PROGRAM MAIN
VAR
	//==============================================================
	// EN: Main machine control function blocks
	// PT: Blocos principais de controle da máquina
	//==============================================================
	instFBSlitter1Control              : FB_SlitterControl;
	instFB_RotaryKnife                 : FB_RotaryKnife;
	// instFB_MetricsAndCalculation    : FB_MetricsAndCalculation;
	instFB_PaperDirectionControl       : FB_PaperDirectionControl;
	instFB_AutomaticOrderChange_V1     : FB_AutomaticOrderChange_V1;
	instFB_AlarmControl                : FB_AlarmControl;
	instFBSavePersistentData           : FB_SavePersistentData;

	//==============================================================
	// EN: Stacker control function blocks
	// PT: Blocos de controle dos empilhadores
	//==============================================================
	instFBLowerStackerControl          : FB_SimpleSheetStackerControl;
	instFBLowerStackerControlV1        : FB_SimpleSheetStackerControl_1;
	instFBUpperStackerControl          : FB_ComplexSheetStackerControl;

	//==============================================================
	// EN: Persistent data control status
	// PT: Estado do controle de dados persistentes
	//==============================================================
	bStart                             : BOOL;
	bError                             : BOOL;
	bBusy                              : BOOL;
	nErrorId                           : UDINT;
	fbR_Trig                           : R_TRIG;

	//==============================================================
	// EN: Machine interlock and control signals
	// PT: Sinais de intertravamento e controle da máquina
	//==============================================================
	slitterHomeComplete                : BOOL;
	aocReferenceSwitch                 : BOOL;
	lineSpeedUpFromAOC                 : BOOL;
	lineSpeedDownFromAOC               : BOOL;
	lineStopFromAOC                    : BOOL;
	executePositioningFromAOC          : BOOL;
	rotaryKnifeSpeedRefFromAOC         : LREAL;
	slitterSpeedRefFromAOC             : LREAL;
	lineStopFromRotaryKnife            : BOOL;
	lineStopFromSlitter                : BOOL;
	lineStopFromLowerStacker           : BOOL;
	aocRunning                         : BOOL;

	//==============================================================
	// EN: Program initialization
	// PT: Inicialização do programa
	//==============================================================
	firstScan                          : BOOL := TRUE;
	lineStopFromUpperStacker: BOOL;
END_VAR

//==============================================================
// EN: Cyclic machine control sequence
// PT: Sequência cíclica de controle da máquina
//==============================================================
_00_UpdateHardware();
_01_SlitterControl();
_02_RotaryKnifeControl();
_04_AutomaticOrderChange();
_05_LineControl();
_06_AlarmsControl();
_07_LowerStackerControl();
_08_UpperStackerControl();

// EN: Publish the upper stacker alarms and include them in the general indication.
// PT: Publica os alarmes do stacker superior e os inclui na indicação geral.
hmiAlarms.upperStacker :=
	instFBUpperStackerControl.hmiAlarms;

hmiStatus.alarmActive :=
	hmiStatus.alarmActive OR
	instFBUpperStackerControl.alarmActive;

// EN: Update persistent data management.
// PT: Atualiza o gerenciamento dos dados persistentes.
instFBSavePersistentData();

// EN: Apply default commands during the first PLC scan.
// PT: Aplica os comandos padrão durante o primeiro ciclo do PLC.
IF firstScan THEN
	hmiCommands.lowerStacker.backstopAutoCmd := TRUE;
	hmiCommands.lowerStacker.conveyorLevelerAutoCmd := TRUE;

	hmiCommands.upperStacker.backstopAutoCmd := TRUE;
	hmiCommands.upperStacker.elevatorAutoCmd := TRUE;

END_IF

firstScan := FALSE;

(*==============================================================================================================================
CPNTeck - Automação industrial
(c)Copyright 2023 All Rights Reserved
_______________________________________________________________________________________________________________________________
Library: <N/A or library name>
Tested with: <PLC / IPC model>
Engineering: <TwinCAT version>
Restrictions: <text>
Requirements: <text>
Functionality: <short description>
Support: <email>
Note: Parameter comments are only available in language 'English (United States)'
_______________________________________________________________________________________________________________________________
Change log table:

Version  		| Date        			| Expert in charge  	| Changes applied
<xx.xx.xx>		| <dd.mm.yyyy>  		| <name>              | <changes>

===============================================================================================================================*)

METHOD _00_UpdateHardware
VAR_INPUT
END_VAR

SLT1_P1_100_UG1();
SLT1_P1_100_UG2();
SLT1_P1_100_UG3();
SLT1_P1_100_UG4();
SLT1_P1_100_UG5();

SLT1_P1_200_UG1();
SLT1_P1_200_UG2();
SLT1_P1_200_UG3();
SLT1_P1_200_UG4();
SLT1_P1_200_UG5();
SLT1_P1_200_UG6();
SLT1_P1_200_UG7();
SLT1_P1_200_UG8();


STK_P2_050_DI1();
STK_P2_050_DI2();
STK_P2_050_DO1();
STK_P2_050_DO2();
	
STK_P2_050_AO1();	
STK_P2_050_AO2();
STK_P2_050_AO3();
STK_P2_050_AO4();

STK_P2_050_ENC1();
//Io-Link master
STK_050_BC2();
//Io-Link Slaves

STKU_050_DIO1();	//Ch 0 - IO-Link IP67 Input/Output module
STKU_050_DIO2(); //Ch 1 - IO-Link DIN Rail Input/Output module
STKU_050_DIO3(); //Ch 1 - IO-Link DIN Rail Input/Output module


STKL_050_DIO1();	//Ch 0 - IO-Link IP67 Input/Output module
STKL_050_DIO2(); //Ch 1 - IO-Link DIN Rail Input/Output module
STKL_100_B01(); //Ch 2 - IO-Link Pile height sensor	

//CANOpen slave	
STKU_P2_100_UG8(enable := TRUE); //Backstop servo drive

// EN: Lift servo drive. Quick stop is generated by the elevator control block.
// PT: Servo do elevador. O quick stop é gerado pelo bloco de controle do elevador.
STKU_P2_100_UG9(enable := TRUE);

// Safety processor (TwinSAFE)
STK_P2_050_SP01(run := TRUE,
				 errorAcknowledgement := hmiCommands.slitter1.resetCmd OR hmiCommands.lowerStacker.resetCmd OR hmiCommands.upperStacker.resetCmd,
				 safetyReset := hmiCommands.slitter1.resetCmd OR hmiCommands.lowerStacker.resetCmd OR hmiCommands.upperStacker.resetCmd
);
END_METHOD

METHOD _01_SlitterControl
VAR_INPUT
END_VAR

//ARK_P1_050_AO02.Channel1
//ARK_P1_050_AO02.Channel3
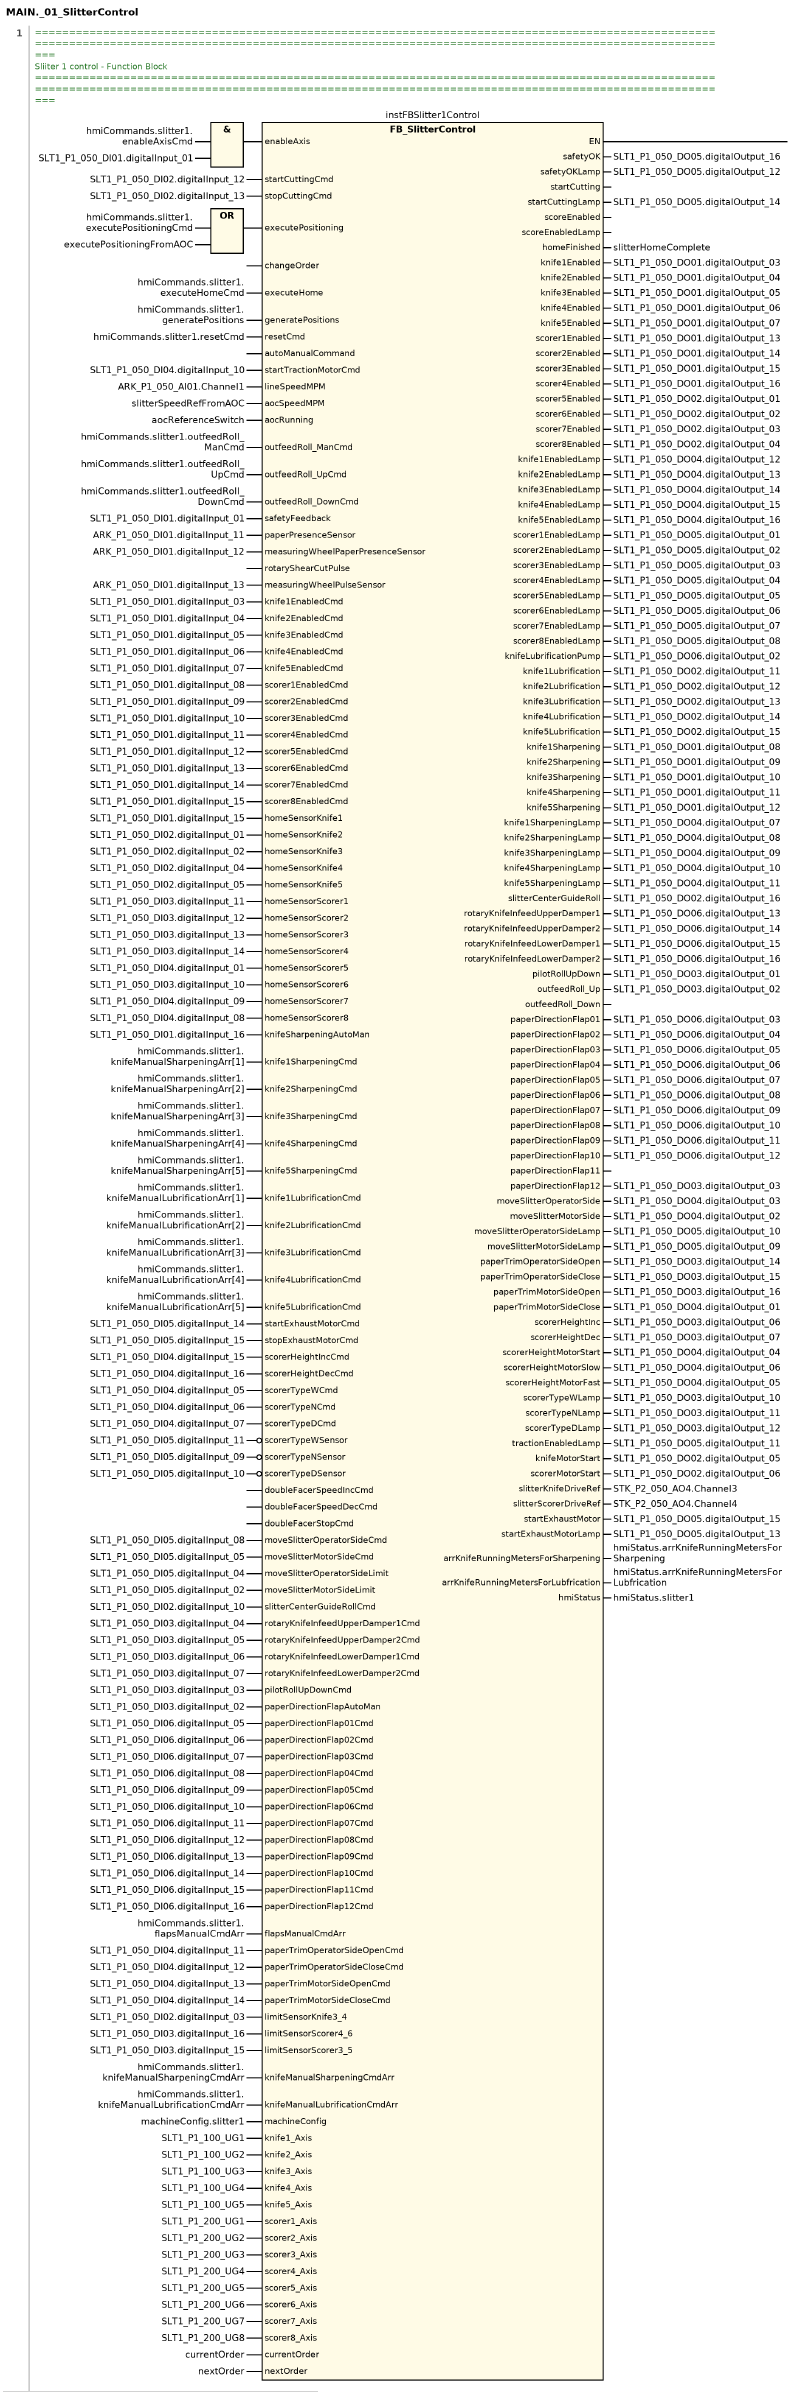
// NETWORK 1
// 					===========================================================================================================================================================================================================
//
// Sliiter 1 control - Function Block
//
// ===========================================================================================================================================================================================================
//
instFBSlitter1Control(
    enableAxis := hmiCommands.slitter1.enableAxisCmd AND SLT1_P1_050_DI01.digitalInput_01,
    startCuttingCmd := SLT1_P1_050_DI02.digitalInput_12,
    stopCuttingCmd := SLT1_P1_050_DI02.digitalInput_13,
    executePositioning := hmiCommands.slitter1.executePositioningCmd OR executePositioningFromAOC,
    executeHome := hmiCommands.slitter1.executeHomeCmd,
    generatePositions := hmiCommands.slitter1.generatePositions,
    resetCmd := hmiCommands.slitter1.resetCmd,
    startTractionMotorCmd := SLT1_P1_050_DI04.digitalInput_10,
    lineSpeedMPM := ARK_P1_050_AI01.Channel1,
    aocSpeedMPM := slitterSpeedRefFromAOC,
    aocRunning := aocReferenceSwitch,
    outfeedRoll_ManCmd := hmiCommands.slitter1.outfeedRoll_ManCmd,
    outfeedRoll_UpCmd := hmiCommands.slitter1.outfeedRoll_UpCmd,
    outfeedRoll_DownCmd := hmiCommands.slitter1.outfeedRoll_DownCmd,
    safetyFeedback := SLT1_P1_050_DI01.digitalInput_01,
    paperPresenceSensor := ARK_P1_050_DI01.digitalInput_11,
    measuringWheelPaperPresenceSensor := ARK_P1_050_DI01.digitalInput_12,
    measuringWheelPulseSensor := ARK_P1_050_DI01.digitalInput_13,
    knife1EnabledCmd := SLT1_P1_050_DI01.digitalInput_03,
    knife2EnabledCmd := SLT1_P1_050_DI01.digitalInput_04,
    knife3EnabledCmd := SLT1_P1_050_DI01.digitalInput_05,
    knife4EnabledCmd := SLT1_P1_050_DI01.digitalInput_06,
    knife5EnabledCmd := SLT1_P1_050_DI01.digitalInput_07,
    scorer1EnabledCmd := SLT1_P1_050_DI01.digitalInput_08,
    scorer2EnabledCmd := SLT1_P1_050_DI01.digitalInput_09,
    scorer3EnabledCmd := SLT1_P1_050_DI01.digitalInput_10,
    scorer4EnabledCmd := SLT1_P1_050_DI01.digitalInput_11,
    scorer5EnabledCmd := SLT1_P1_050_DI01.digitalInput_12,
    scorer6EnabledCmd := SLT1_P1_050_DI01.digitalInput_13,
    scorer7EnabledCmd := SLT1_P1_050_DI01.digitalInput_14,
    scorer8EnabledCmd := SLT1_P1_050_DI01.digitalInput_15,
    homeSensorKnife1 := SLT1_P1_050_DI01.digitalInput_15,
    homeSensorKnife2 := SLT1_P1_050_DI02.digitalInput_01,
    homeSensorKnife3 := SLT1_P1_050_DI02.digitalInput_02,
    homeSensorKnife4 := SLT1_P1_050_DI02.digitalInput_04,
    homeSensorKnife5 := SLT1_P1_050_DI02.digitalInput_05,
    homeSensorScorer1 := SLT1_P1_050_DI03.digitalInput_11,
    homeSensorScorer2 := SLT1_P1_050_DI03.digitalInput_12,
    homeSensorScorer3 := SLT1_P1_050_DI03.digitalInput_13,
    homeSensorScorer4 := SLT1_P1_050_DI03.digitalInput_14,
    homeSensorScorer5 := SLT1_P1_050_DI04.digitalInput_01,
    homeSensorScorer6 := SLT1_P1_050_DI03.digitalInput_10,
    homeSensorScorer7 := SLT1_P1_050_DI04.digitalInput_09,
    homeSensorScorer8 := SLT1_P1_050_DI04.digitalInput_08,
    knifeSharpeningAutoMan := SLT1_P1_050_DI01.digitalInput_16,
    knife1SharpeningCmd := hmiCommands.slitter1.knifeManualSharpeningArr[1],
    knife2SharpeningCmd := hmiCommands.slitter1.knifeManualSharpeningArr[2],
    knife3SharpeningCmd := hmiCommands.slitter1.knifeManualSharpeningArr[3],
    knife4SharpeningCmd := hmiCommands.slitter1.knifeManualSharpeningArr[4],
    knife5SharpeningCmd := hmiCommands.slitter1.knifeManualSharpeningArr[5],
    knife1LubrificationCmd := hmiCommands.slitter1.knifeManualLubrificationArr[1],
    knife2LubrificationCmd := hmiCommands.slitter1.knifeManualLubrificationArr[2],
    knife3LubrificationCmd := hmiCommands.slitter1.knifeManualLubrificationArr[3],
    knife4LubrificationCmd := hmiCommands.slitter1.knifeManualLubrificationArr[4],
    knife5LubrificationCmd := hmiCommands.slitter1.knifeManualLubrificationArr[5],
    startExhaustMotorCmd := SLT1_P1_050_DI05.digitalInput_14,
    stopExhaustMotorCmd := SLT1_P1_050_DI05.digitalInput_15,
    scorerHeightIncCmd := SLT1_P1_050_DI04.digitalInput_15,
    scorerHeightDecCmd := SLT1_P1_050_DI04.digitalInput_16,
    scorerTypeWCmd := SLT1_P1_050_DI04.digitalInput_05,
    scorerTypeNCmd := SLT1_P1_050_DI04.digitalInput_06,
    scorerTypeDCmd := SLT1_P1_050_DI04.digitalInput_07,
    scorerTypeWSensor := NOT SLT1_P1_050_DI05.digitalInput_11,
    scorerTypeNSensor := NOT SLT1_P1_050_DI05.digitalInput_09,
    scorerTypeDSensor := NOT SLT1_P1_050_DI05.digitalInput_10,
    moveSlitterOperatorSideCmd := SLT1_P1_050_DI05.digitalInput_08,
    moveSlitterMotorSideCmd := SLT1_P1_050_DI05.digitalInput_05,
    moveSlitterOperatorSideLimit := SLT1_P1_050_DI05.digitalInput_04,
    moveSlitterMotorSideLimit := SLT1_P1_050_DI05.digitalInput_02,
    slitterCenterGuideRollCmd := SLT1_P1_050_DI02.digitalInput_10,
    rotaryKnifeInfeedUpperDamper1Cmd := SLT1_P1_050_DI03.digitalInput_04,
    rotaryKnifeInfeedUpperDamper2Cmd := SLT1_P1_050_DI03.digitalInput_05,
    rotaryKnifeInfeedLowerDamper1Cmd := SLT1_P1_050_DI03.digitalInput_06,
    rotaryKnifeInfeedLowerDamper2Cmd := SLT1_P1_050_DI03.digitalInput_07,
    pilotRollUpDownCmd := SLT1_P1_050_DI03.digitalInput_03,
    paperDirectionFlapAutoMan := SLT1_P1_050_DI03.digitalInput_02,
    paperDirectionFlap01Cmd := SLT1_P1_050_DI06.digitalInput_05,
    paperDirectionFlap02Cmd := SLT1_P1_050_DI06.digitalInput_06,
    paperDirectionFlap03Cmd := SLT1_P1_050_DI06.digitalInput_07,
    paperDirectionFlap04Cmd := SLT1_P1_050_DI06.digitalInput_08,
    paperDirectionFlap05Cmd := SLT1_P1_050_DI06.digitalInput_09,
    paperDirectionFlap06Cmd := SLT1_P1_050_DI06.digitalInput_10,
    paperDirectionFlap07Cmd := SLT1_P1_050_DI06.digitalInput_11,
    paperDirectionFlap08Cmd := SLT1_P1_050_DI06.digitalInput_12,
    paperDirectionFlap09Cmd := SLT1_P1_050_DI06.digitalInput_13,
    paperDirectionFlap10Cmd := SLT1_P1_050_DI06.digitalInput_14,
    paperDirectionFlap11Cmd := SLT1_P1_050_DI06.digitalInput_15,
    paperDirectionFlap12Cmd := SLT1_P1_050_DI06.digitalInput_16,
    flapsManualCmdArr := hmiCommands.slitter1.flapsManualCmdArr,
    paperTrimOperatorSideOpenCmd := SLT1_P1_050_DI04.digitalInput_11,
    paperTrimOperatorSideCloseCmd := SLT1_P1_050_DI04.digitalInput_12,
    paperTrimMotorSideOpenCmd := SLT1_P1_050_DI04.digitalInput_13,
    paperTrimMotorSideCloseCmd := SLT1_P1_050_DI04.digitalInput_14,
    limitSensorKnife3_4 := SLT1_P1_050_DI02.digitalInput_03,
    limitSensorScorer4_6 := SLT1_P1_050_DI03.digitalInput_16,
    limitSensorScorer3_5 := SLT1_P1_050_DI03.digitalInput_15,
    knifeManualSharpeningCmdArr := hmiCommands.slitter1.knifeManualSharpeningCmdArr,
    knifeManualLubrificationCmdArr := hmiCommands.slitter1.knifeManualLubrificationCmdArr,
    machineConfig := machineConfig.slitter1,
    knife1_Axis := SLT1_P1_100_UG1,
    knife2_Axis := SLT1_P1_100_UG2,
    knife3_Axis := SLT1_P1_100_UG3,
    knife4_Axis := SLT1_P1_100_UG4,
    knife5_Axis := SLT1_P1_100_UG5,
    scorer1_Axis := SLT1_P1_200_UG1,
    scorer2_Axis := SLT1_P1_200_UG2,
    scorer3_Axis := SLT1_P1_200_UG3,
    scorer4_Axis := SLT1_P1_200_UG4,
    scorer5_Axis := SLT1_P1_200_UG5,
    scorer6_Axis := SLT1_P1_200_UG6,
    scorer7_Axis := SLT1_P1_200_UG7,
    scorer8_Axis := SLT1_P1_200_UG8,
    currentOrder := currentOrder,
    nextOrder := nextOrder,
    safetyOK => SLT1_P1_050_DO05.digitalOutput_16,
    safetyOKLamp => SLT1_P1_050_DO05.digitalOutput_12,
    startCuttingLamp => SLT1_P1_050_DO05.digitalOutput_14,
    homeFinished => slitterHomeComplete,
    knife1Enabled => SLT1_P1_050_DO01.digitalOutput_03,
    knife2Enabled => SLT1_P1_050_DO01.digitalOutput_04,
    knife3Enabled => SLT1_P1_050_DO01.digitalOutput_05,
    knife4Enabled => SLT1_P1_050_DO01.digitalOutput_06,
    knife5Enabled => SLT1_P1_050_DO01.digitalOutput_07,
    scorer1Enabled => SLT1_P1_050_DO01.digitalOutput_13,
    scorer2Enabled => SLT1_P1_050_DO01.digitalOutput_14,
    scorer3Enabled => SLT1_P1_050_DO01.digitalOutput_15,
    scorer4Enabled => SLT1_P1_050_DO01.digitalOutput_16,
    scorer5Enabled => SLT1_P1_050_DO02.digitalOutput_01,
    scorer6Enabled => SLT1_P1_050_DO02.digitalOutput_02,
    scorer7Enabled => SLT1_P1_050_DO02.digitalOutput_03,
    scorer8Enabled => SLT1_P1_050_DO02.digitalOutput_04,
    knife1EnabledLamp => SLT1_P1_050_DO04.digitalOutput_12,
    knife2EnabledLamp => SLT1_P1_050_DO04.digitalOutput_13,
    knife3EnabledLamp => SLT1_P1_050_DO04.digitalOutput_14,
    knife4EnabledLamp => SLT1_P1_050_DO04.digitalOutput_15,
    knife5EnabledLamp => SLT1_P1_050_DO04.digitalOutput_16,
    scorer1EnabledLamp => SLT1_P1_050_DO05.digitalOutput_01,
    scorer2EnabledLamp => SLT1_P1_050_DO05.digitalOutput_02,
    scorer3EnabledLamp => SLT1_P1_050_DO05.digitalOutput_03,
    scorer4EnabledLamp => SLT1_P1_050_DO05.digitalOutput_04,
    scorer5EnabledLamp => SLT1_P1_050_DO05.digitalOutput_05,
    scorer6EnabledLamp => SLT1_P1_050_DO05.digitalOutput_06,
    scorer7EnabledLamp => SLT1_P1_050_DO05.digitalOutput_07,
    scorer8EnabledLamp => SLT1_P1_050_DO05.digitalOutput_08,
    knifeLubrificationPump => SLT1_P1_050_DO06.digitalOutput_02,
    knife1Lubrification => SLT1_P1_050_DO02.digitalOutput_11,
    knife2Lubrification => SLT1_P1_050_DO02.digitalOutput_12,
    knife3Lubrification => SLT1_P1_050_DO02.digitalOutput_13,
    knife4Lubrification => SLT1_P1_050_DO02.digitalOutput_14,
    knife5Lubrification => SLT1_P1_050_DO02.digitalOutput_15,
    knife1Sharpening => SLT1_P1_050_DO01.digitalOutput_08,
    knife2Sharpening => SLT1_P1_050_DO01.digitalOutput_09,
    knife3Sharpening => SLT1_P1_050_DO01.digitalOutput_10,
    knife4Sharpening => SLT1_P1_050_DO01.digitalOutput_11,
    knife5Sharpening => SLT1_P1_050_DO01.digitalOutput_12,
    knife1SharpeningLamp => SLT1_P1_050_DO04.digitalOutput_07,
    knife2SharpeningLamp => SLT1_P1_050_DO04.digitalOutput_08,
    knife3SharpeningLamp => SLT1_P1_050_DO04.digitalOutput_09,
    knife4SharpeningLamp => SLT1_P1_050_DO04.digitalOutput_10,
    knife5SharpeningLamp => SLT1_P1_050_DO04.digitalOutput_11,
    slitterCenterGuideRoll => SLT1_P1_050_DO02.digitalOutput_16,
    rotaryKnifeInfeedUpperDamper1 => SLT1_P1_050_DO06.digitalOutput_13,
    rotaryKnifeInfeedUpperDamper2 => SLT1_P1_050_DO06.digitalOutput_14,
    rotaryKnifeInfeedLowerDamper1 => SLT1_P1_050_DO06.digitalOutput_15,
    rotaryKnifeInfeedLowerDamper2 => SLT1_P1_050_DO06.digitalOutput_16,
    pilotRollUpDown => SLT1_P1_050_DO03.digitalOutput_01,
    outfeedRoll_Up => SLT1_P1_050_DO03.digitalOutput_02,
    paperDirectionFlap01 => SLT1_P1_050_DO06.digitalOutput_03,
    paperDirectionFlap02 => SLT1_P1_050_DO06.digitalOutput_04,
    paperDirectionFlap03 => SLT1_P1_050_DO06.digitalOutput_05,
    paperDirectionFlap04 => SLT1_P1_050_DO06.digitalOutput_06,
    paperDirectionFlap05 => SLT1_P1_050_DO06.digitalOutput_07,
    paperDirectionFlap06 => SLT1_P1_050_DO06.digitalOutput_08,
    paperDirectionFlap07 => SLT1_P1_050_DO06.digitalOutput_09,
    paperDirectionFlap08 => SLT1_P1_050_DO06.digitalOutput_10,
    paperDirectionFlap09 => SLT1_P1_050_DO06.digitalOutput_11,
    paperDirectionFlap10 => SLT1_P1_050_DO06.digitalOutput_12,
    paperDirectionFlap12 => SLT1_P1_050_DO03.digitalOutput_03,
    moveSlitterOperatorSide => SLT1_P1_050_DO04.digitalOutput_03,
    moveSlitterMotorSide => SLT1_P1_050_DO04.digitalOutput_02,
    moveSlitterOperatorSideLamp => SLT1_P1_050_DO05.digitalOutput_10,
    moveSlitterMotorSideLamp => SLT1_P1_050_DO05.digitalOutput_09,
    paperTrimOperatorSideOpen => SLT1_P1_050_DO03.digitalOutput_14,
    paperTrimOperatorSideClose => SLT1_P1_050_DO03.digitalOutput_15,
    paperTrimMotorSideOpen => SLT1_P1_050_DO03.digitalOutput_16,
    paperTrimMotorSideClose => SLT1_P1_050_DO04.digitalOutput_01,
    scorerHeightInc => SLT1_P1_050_DO03.digitalOutput_06,
    scorerHeightDec => SLT1_P1_050_DO03.digitalOutput_07,
    scorerHeightMotorStart => SLT1_P1_050_DO04.digitalOutput_04,
    scorerHeightMotorSlow => SLT1_P1_050_DO04.digitalOutput_06,
    scorerHeightMotorFast => SLT1_P1_050_DO04.digitalOutput_05,
    scorerTypeWLamp => SLT1_P1_050_DO03.digitalOutput_10,
    scorerTypeNLamp => SLT1_P1_050_DO03.digitalOutput_11,
    scorerTypeDLamp => SLT1_P1_050_DO03.digitalOutput_12,
    tractionEnabledLamp => SLT1_P1_050_DO05.digitalOutput_11,
    knifeMotorStart => SLT1_P1_050_DO02.digitalOutput_05,
    scorerMotorStart => SLT1_P1_050_DO02.digitalOutput_06,
    slitterKnifeDriveRef => STK_P2_050_AO4.Channel3,
    slitterScorerDriveRef => STK_P2_050_AO4.Channel4,
    startExhaustMotor => SLT1_P1_050_DO05.digitalOutput_15,
    startExhaustMotorLamp => SLT1_P1_050_DO05.digitalOutput_13,
    arrKnifeRunningMetersForSharpening => hmiStatus.arrKnifeRunningMetersForSharpening,
    arrKnifeRunningMetersForLubfrication => hmiStatus.arrKnifeRunningMetersForLubfrication,
    hmiStatus => hmiStatus.slitter1); // FB_SlitterControl
END_METHOD

METHOD _02_RotaryKnifeControl
VAR_INPUT
END_VAR

(*


ARK_050_DI01.digitalInput_01 => exitGuardOpen
ARK_050_DI01.digitalInput_02 => lowerKnifeGuardClosed
ARK_050_DI01.digitalInput_03 => upperKnifeGuardClosed
ARK_050_DI01.digitalInput_04 => infeedGuardOpen

ARK_050_DI01.digitalInput_05 => lowerOilLevelLow
ARK_050_DI01.digitalInput_06 => upperOilLevelLow
ARK_050_DI01.digitalInput_07 => exhaustPressurized
ARK_050_DI01.digitalInput_08 => exhaustDepressurized

ARK_050_DI01.digitalInput_09 => upperLevelPaperSensor
ARK_050_DI01.digitalInput_10 => upperKnifeJamDetected
ARK_050_DI01.digitalInput_11 => lowerLevelPaperSensor
ARK_050_DI01.digitalInput_12 => lowerKnifeJamDetected

ARK_050_DI01.digitalInput_13 => lowerKnifeHome
ARK_050_DI01.digitalInput_14 => upperKnifeHome

*)
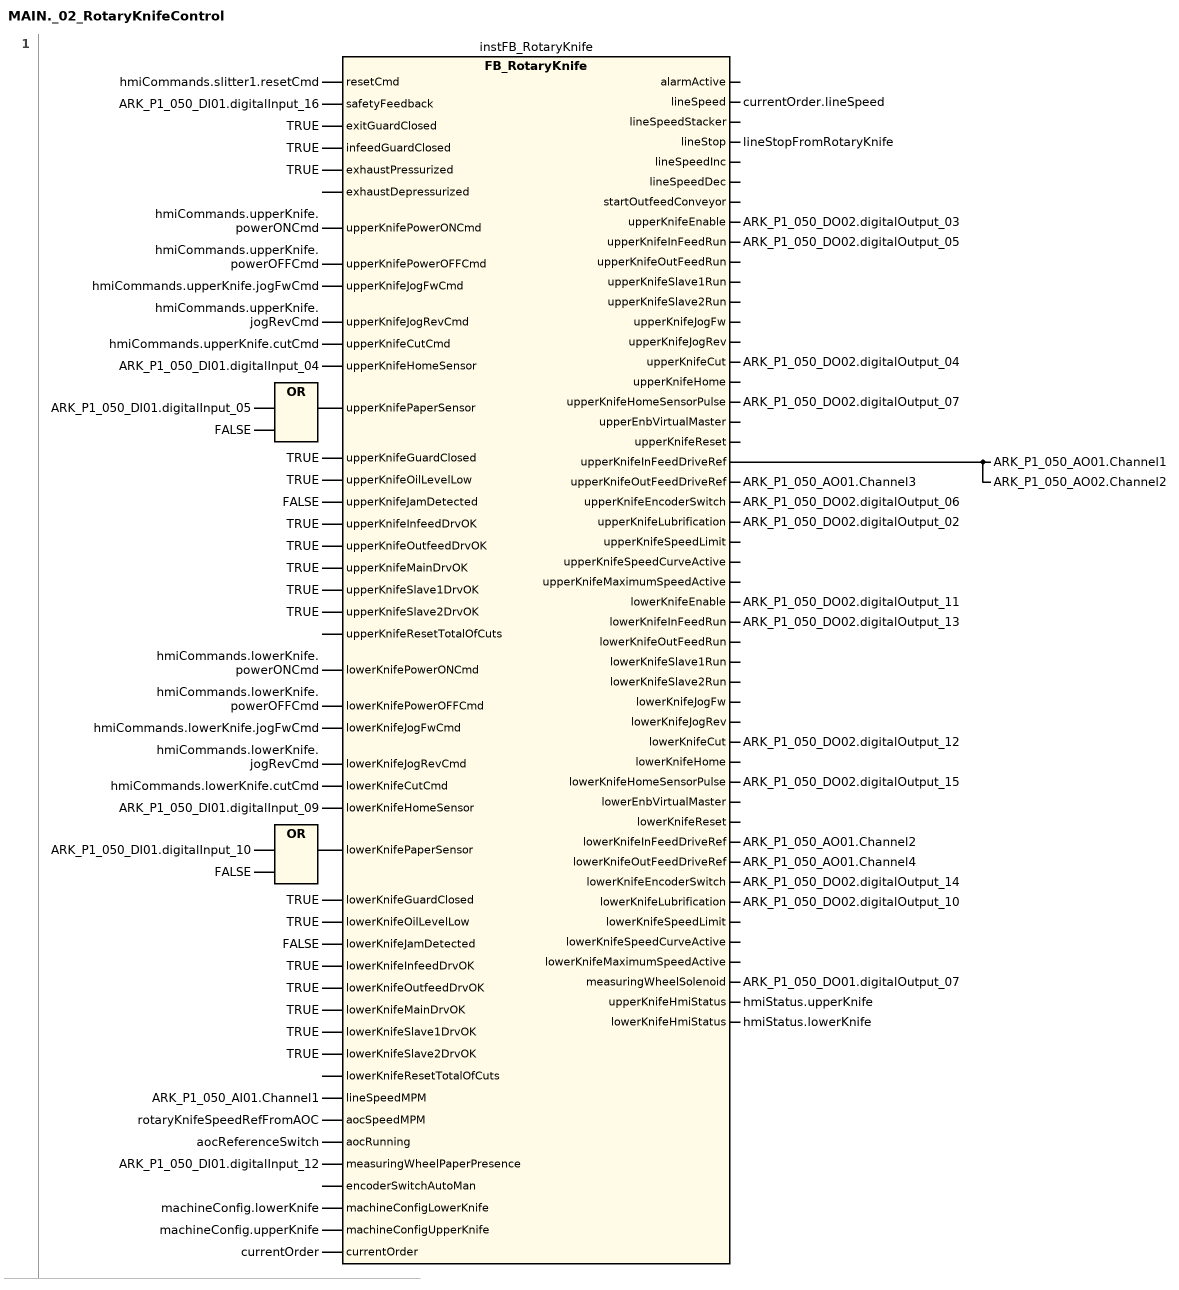
// NETWORK 1
instFB_RotaryKnife(
    resetCmd := hmiCommands.slitter1.resetCmd,
    safetyFeedback := ARK_P1_050_DI01.digitalInput_16,
    exitGuardClosed := TRUE,
    infeedGuardClosed := TRUE,
    exhaustPressurized := TRUE,
    upperKnifePowerONCmd := hmiCommands.upperKnife.powerONCmd,
    upperKnifePowerOFFCmd := hmiCommands.upperKnife.powerOFFCmd,
    upperKnifeJogFwCmd := hmiCommands.upperKnife.jogFwCmd,
    upperKnifeJogRevCmd := hmiCommands.upperKnife.jogRevCmd,
    upperKnifeCutCmd := hmiCommands.upperKnife.cutCmd,
    upperKnifeHomeSensor := ARK_P1_050_DI01.digitalInput_04,
    upperKnifePaperSensor := ARK_P1_050_DI01.digitalInput_05 OR FALSE,
    upperKnifeGuardClosed := TRUE,
    upperKnifeOilLevelLow := TRUE,
    upperKnifeJamDetected := FALSE,
    upperKnifeInfeedDrvOK := TRUE,
    upperKnifeOutfeedDrvOK := TRUE,
    upperKnifeMainDrvOK := TRUE,
    upperKnifeSlave1DrvOK := TRUE,
    upperKnifeSlave2DrvOK := TRUE,
    lowerKnifePowerONCmd := hmiCommands.lowerKnife.powerONCmd,
    lowerKnifePowerOFFCmd := hmiCommands.lowerKnife.powerOFFCmd,
    lowerKnifeJogFwCmd := hmiCommands.lowerKnife.jogFwCmd,
    lowerKnifeJogRevCmd := hmiCommands.lowerKnife.jogRevCmd,
    lowerKnifeCutCmd := hmiCommands.lowerKnife.cutCmd,
    lowerKnifeHomeSensor := ARK_P1_050_DI01.digitalInput_09,
    lowerKnifePaperSensor := ARK_P1_050_DI01.digitalInput_10 OR FALSE,
    lowerKnifeGuardClosed := TRUE,
    lowerKnifeOilLevelLow := TRUE,
    lowerKnifeJamDetected := FALSE,
    lowerKnifeInfeedDrvOK := TRUE,
    lowerKnifeOutfeedDrvOK := TRUE,
    lowerKnifeMainDrvOK := TRUE,
    lowerKnifeSlave1DrvOK := TRUE,
    lowerKnifeSlave2DrvOK := TRUE,
    lineSpeedMPM := ARK_P1_050_AI01.Channel1,
    aocSpeedMPM := rotaryKnifeSpeedRefFromAOC,
    aocRunning := aocReferenceSwitch,
    measuringWheelPaperPresence := ARK_P1_050_DI01.digitalInput_12,
    machineConfigLowerKnife := machineConfig.lowerKnife,
    machineConfigUpperKnife := machineConfig.upperKnife,
    currentOrder := currentOrder,
    lineSpeed => currentOrder.lineSpeed,
    lineStop => lineStopFromRotaryKnife,
    upperKnifeEnable => ARK_P1_050_DO02.digitalOutput_03,
    upperKnifeInFeedRun => ARK_P1_050_DO02.digitalOutput_05,
    upperKnifeCut => ARK_P1_050_DO02.digitalOutput_04,
    upperKnifeHomeSensorPulse => ARK_P1_050_DO02.digitalOutput_07,
    upperKnifeOutFeedDriveRef => ARK_P1_050_AO01.Channel3,
    upperKnifeEncoderSwitch => ARK_P1_050_DO02.digitalOutput_06,
    upperKnifeLubrification => ARK_P1_050_DO02.digitalOutput_02,
    lowerKnifeEnable => ARK_P1_050_DO02.digitalOutput_11,
    lowerKnifeInFeedRun => ARK_P1_050_DO02.digitalOutput_13,
    lowerKnifeCut => ARK_P1_050_DO02.digitalOutput_12,
    lowerKnifeHomeSensorPulse => ARK_P1_050_DO02.digitalOutput_15,
    lowerKnifeInFeedDriveRef => ARK_P1_050_AO01.Channel2,
    lowerKnifeOutFeedDriveRef => ARK_P1_050_AO01.Channel4,
    lowerKnifeEncoderSwitch => ARK_P1_050_DO02.digitalOutput_14,
    lowerKnifeLubrification => ARK_P1_050_DO02.digitalOutput_10,
    measuringWheelSolenoid => ARK_P1_050_DO01.digitalOutput_07,
    upperKnifeHmiStatus => hmiStatus.upperKnife,
    lowerKnifeHmiStatus => hmiStatus.lowerKnife); // FB_RotaryKnife
ARK_P1_050_AO01.Channel1 := instFB_RotaryKnife.upperKnifeInFeedDriveRef;
ARK_P1_050_AO02.Channel2 := instFB_RotaryKnife.upperKnifeInFeedDriveRef;
END_METHOD

METHOD _04_AutomaticOrderChange
VAR_INPUT
END_VAR
(*

	SLT1_C1_050_DI01     : FB_EL1809;        // Digital inputs card
    SLT1_C1_050_DO01     : FB_EL2809;        // Digital outputs card

*)
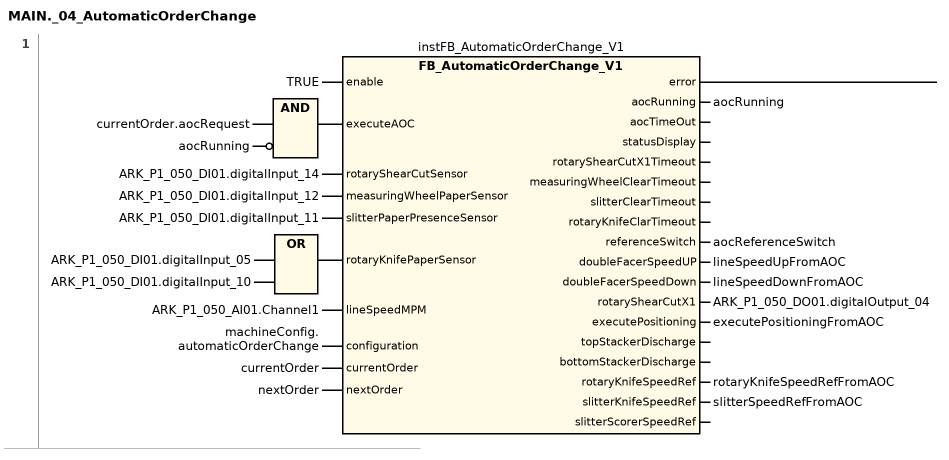
// NETWORK 1
instFB_AutomaticOrderChange_V1(
    enable := TRUE,
    executeAOC := currentOrder.aocRequest AND NOT aocRunning,
    rotaryShearCutSensor := ARK_P1_050_DI01.digitalInput_14,
    measuringWheelPaperSensor := ARK_P1_050_DI01.digitalInput_12,
    slitterPaperPresenceSensor := ARK_P1_050_DI01.digitalInput_11,
    rotaryKnifePaperSensor := ARK_P1_050_DI01.digitalInput_05 OR ARK_P1_050_DI01.digitalInput_10,
    lineSpeedMPM := ARK_P1_050_AI01.Channel1,
    configuration := machineConfig.automaticOrderChange,
    currentOrder := currentOrder,
    nextOrder := nextOrder,
    aocRunning => aocRunning,
    referenceSwitch => aocReferenceSwitch,
    doubleFacerSpeedUP => lineSpeedUpFromAOC,
    doubleFacerSpeedDown => lineSpeedDownFromAOC,
    rotaryShearCutX1 => ARK_P1_050_DO01.digitalOutput_04,
    executePositioning => executePositioningFromAOC,
    rotaryKnifeSpeedRef => rotaryKnifeSpeedRefFromAOC,
    slitterKnifeSpeedRef => slitterSpeedRefFromAOC); // FB_AutomaticOrderChange_V1
END_METHOD

METHOD _05_LineControl
VAR_INPUT
END_VAR
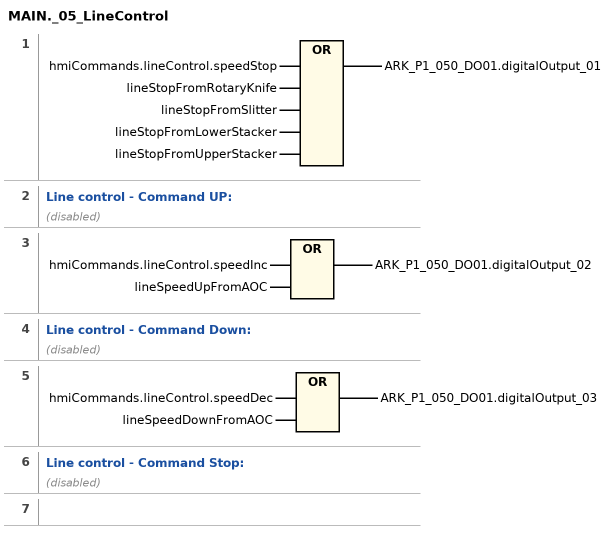
// NETWORK 1
ARK_P1_050_DO01.digitalOutput_01 := hmiCommands.lineControl.speedStop OR lineStopFromRotaryKnife OR lineStopFromSlitter OR lineStopFromLowerStacker OR lineStopFromUpperStacker;

// NETWORK 2 (disabled)
// label: Line control - Command UP

// NETWORK 3
ARK_P1_050_DO01.digitalOutput_02 := hmiCommands.lineControl.speedInc OR lineSpeedUpFromAOC;

// NETWORK 4 (disabled)
// label: Line control - Command Down

// NETWORK 5
ARK_P1_050_DO01.digitalOutput_03 := hmiCommands.lineControl.speedDec OR lineSpeedDownFromAOC;

// NETWORK 6 (disabled)
// label: Line control - Command Stop

// NETWORK 7
END_METHOD

METHOD _06_AlarmsControl
VAR_INPUT
END_VAR
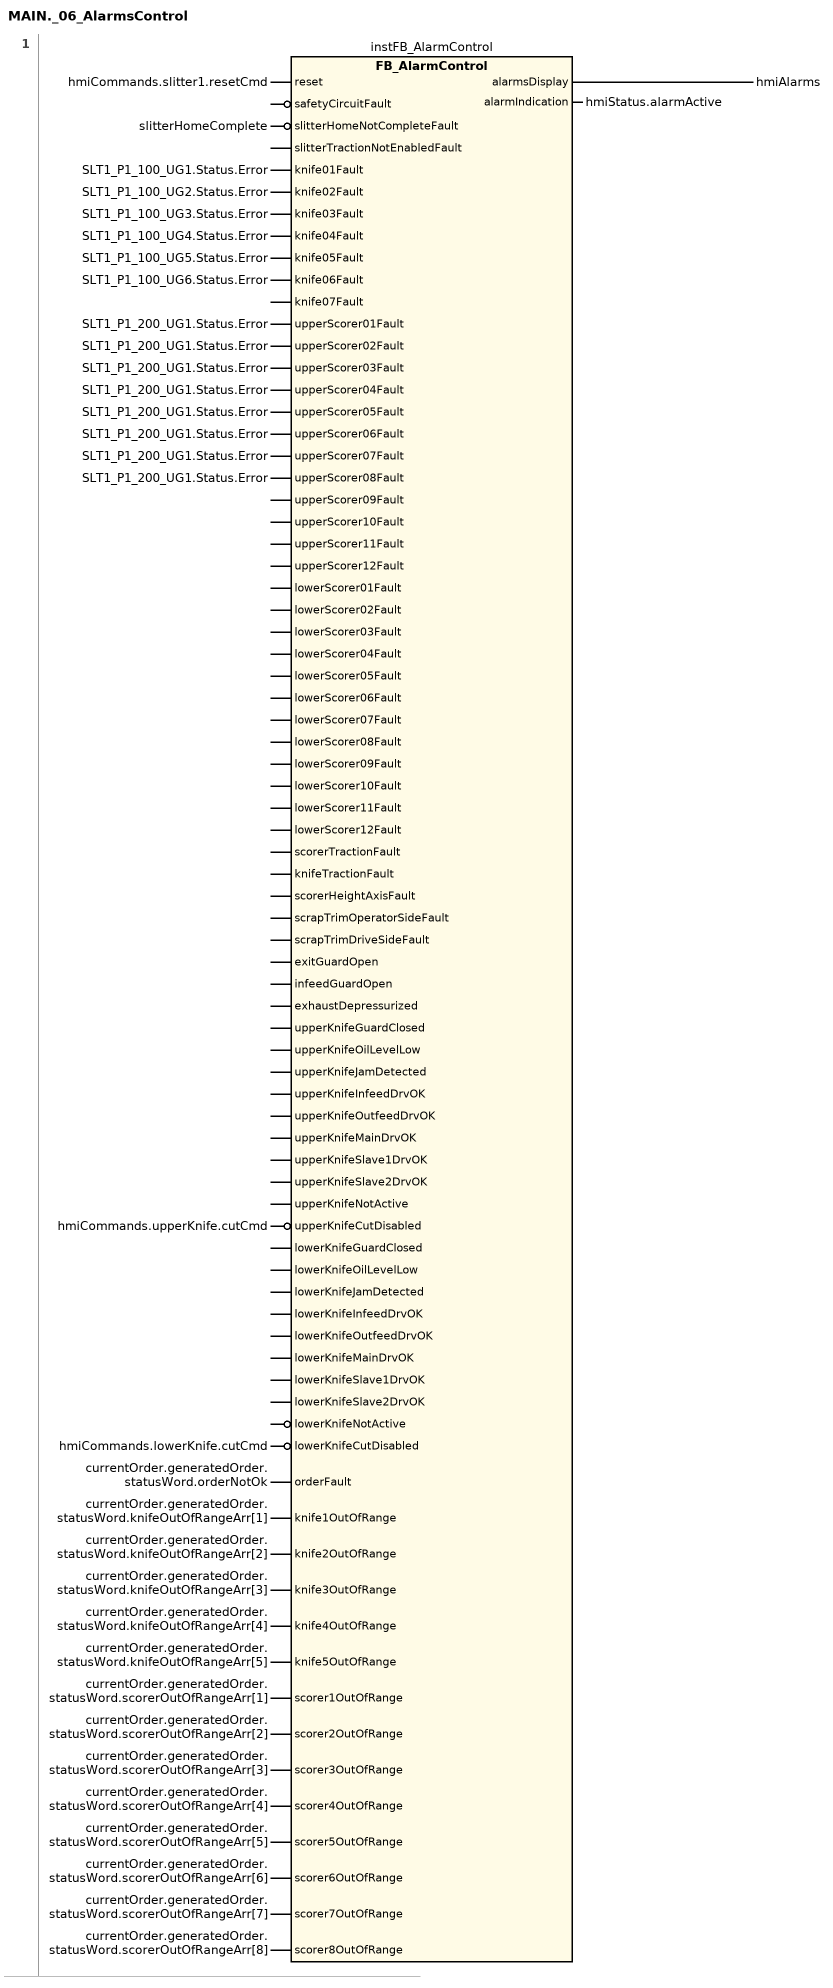
// NETWORK 1
instFB_AlarmControl(
    reset := hmiCommands.slitter1.resetCmd,
    slitterHomeNotCompleteFault := NOT slitterHomeComplete,
    knife01Fault := SLT1_P1_100_UG1.Status.Error,
    knife02Fault := SLT1_P1_100_UG2.Status.Error,
    knife03Fault := SLT1_P1_100_UG3.Status.Error,
    knife04Fault := SLT1_P1_100_UG4.Status.Error,
    knife05Fault := SLT1_P1_100_UG5.Status.Error,
    knife06Fault := SLT1_P1_100_UG6.Status.Error,
    upperScorer01Fault := SLT1_P1_200_UG1.Status.Error,
    upperScorer02Fault := SLT1_P1_200_UG1.Status.Error,
    upperScorer03Fault := SLT1_P1_200_UG1.Status.Error,
    upperScorer04Fault := SLT1_P1_200_UG1.Status.Error,
    upperScorer05Fault := SLT1_P1_200_UG1.Status.Error,
    upperScorer06Fault := SLT1_P1_200_UG1.Status.Error,
    upperScorer07Fault := SLT1_P1_200_UG1.Status.Error,
    upperScorer08Fault := SLT1_P1_200_UG1.Status.Error,
    upperKnifeCutDisabled := NOT hmiCommands.upperKnife.cutCmd,
    lowerKnifeCutDisabled := NOT hmiCommands.lowerKnife.cutCmd,
    orderFault := currentOrder.generatedOrder.statusWord.orderNotOk,
    knife1OutOfRange := currentOrder.generatedOrder.statusWord.knifeOutOfRangeArr[1],
    knife2OutOfRange := currentOrder.generatedOrder.statusWord.knifeOutOfRangeArr[2],
    knife3OutOfRange := currentOrder.generatedOrder.statusWord.knifeOutOfRangeArr[3],
    knife4OutOfRange := currentOrder.generatedOrder.statusWord.knifeOutOfRangeArr[4],
    knife5OutOfRange := currentOrder.generatedOrder.statusWord.knifeOutOfRangeArr[5],
    scorer1OutOfRange := currentOrder.generatedOrder.statusWord.scorerOutOfRangeArr[1],
    scorer2OutOfRange := currentOrder.generatedOrder.statusWord.scorerOutOfRangeArr[2],
    scorer3OutOfRange := currentOrder.generatedOrder.statusWord.scorerOutOfRangeArr[3],
    scorer4OutOfRange := currentOrder.generatedOrder.statusWord.scorerOutOfRangeArr[4],
    scorer5OutOfRange := currentOrder.generatedOrder.statusWord.scorerOutOfRangeArr[5],
    scorer6OutOfRange := currentOrder.generatedOrder.statusWord.scorerOutOfRangeArr[6],
    scorer7OutOfRange := currentOrder.generatedOrder.statusWord.scorerOutOfRangeArr[7],
    scorer8OutOfRange := currentOrder.generatedOrder.statusWord.scorerOutOfRangeArr[8],
    alarmIndication => hmiStatus.alarmActive); // FB_AlarmControl
hmiAlarms := instFB_AlarmControl.alarmsDisplay;
END_METHOD

METHOD _07_LowerStackerControl
VAR_INPUT
END_VAR

VAR
	
//ARK_P1_050_AO01.Channel2
END_VAR
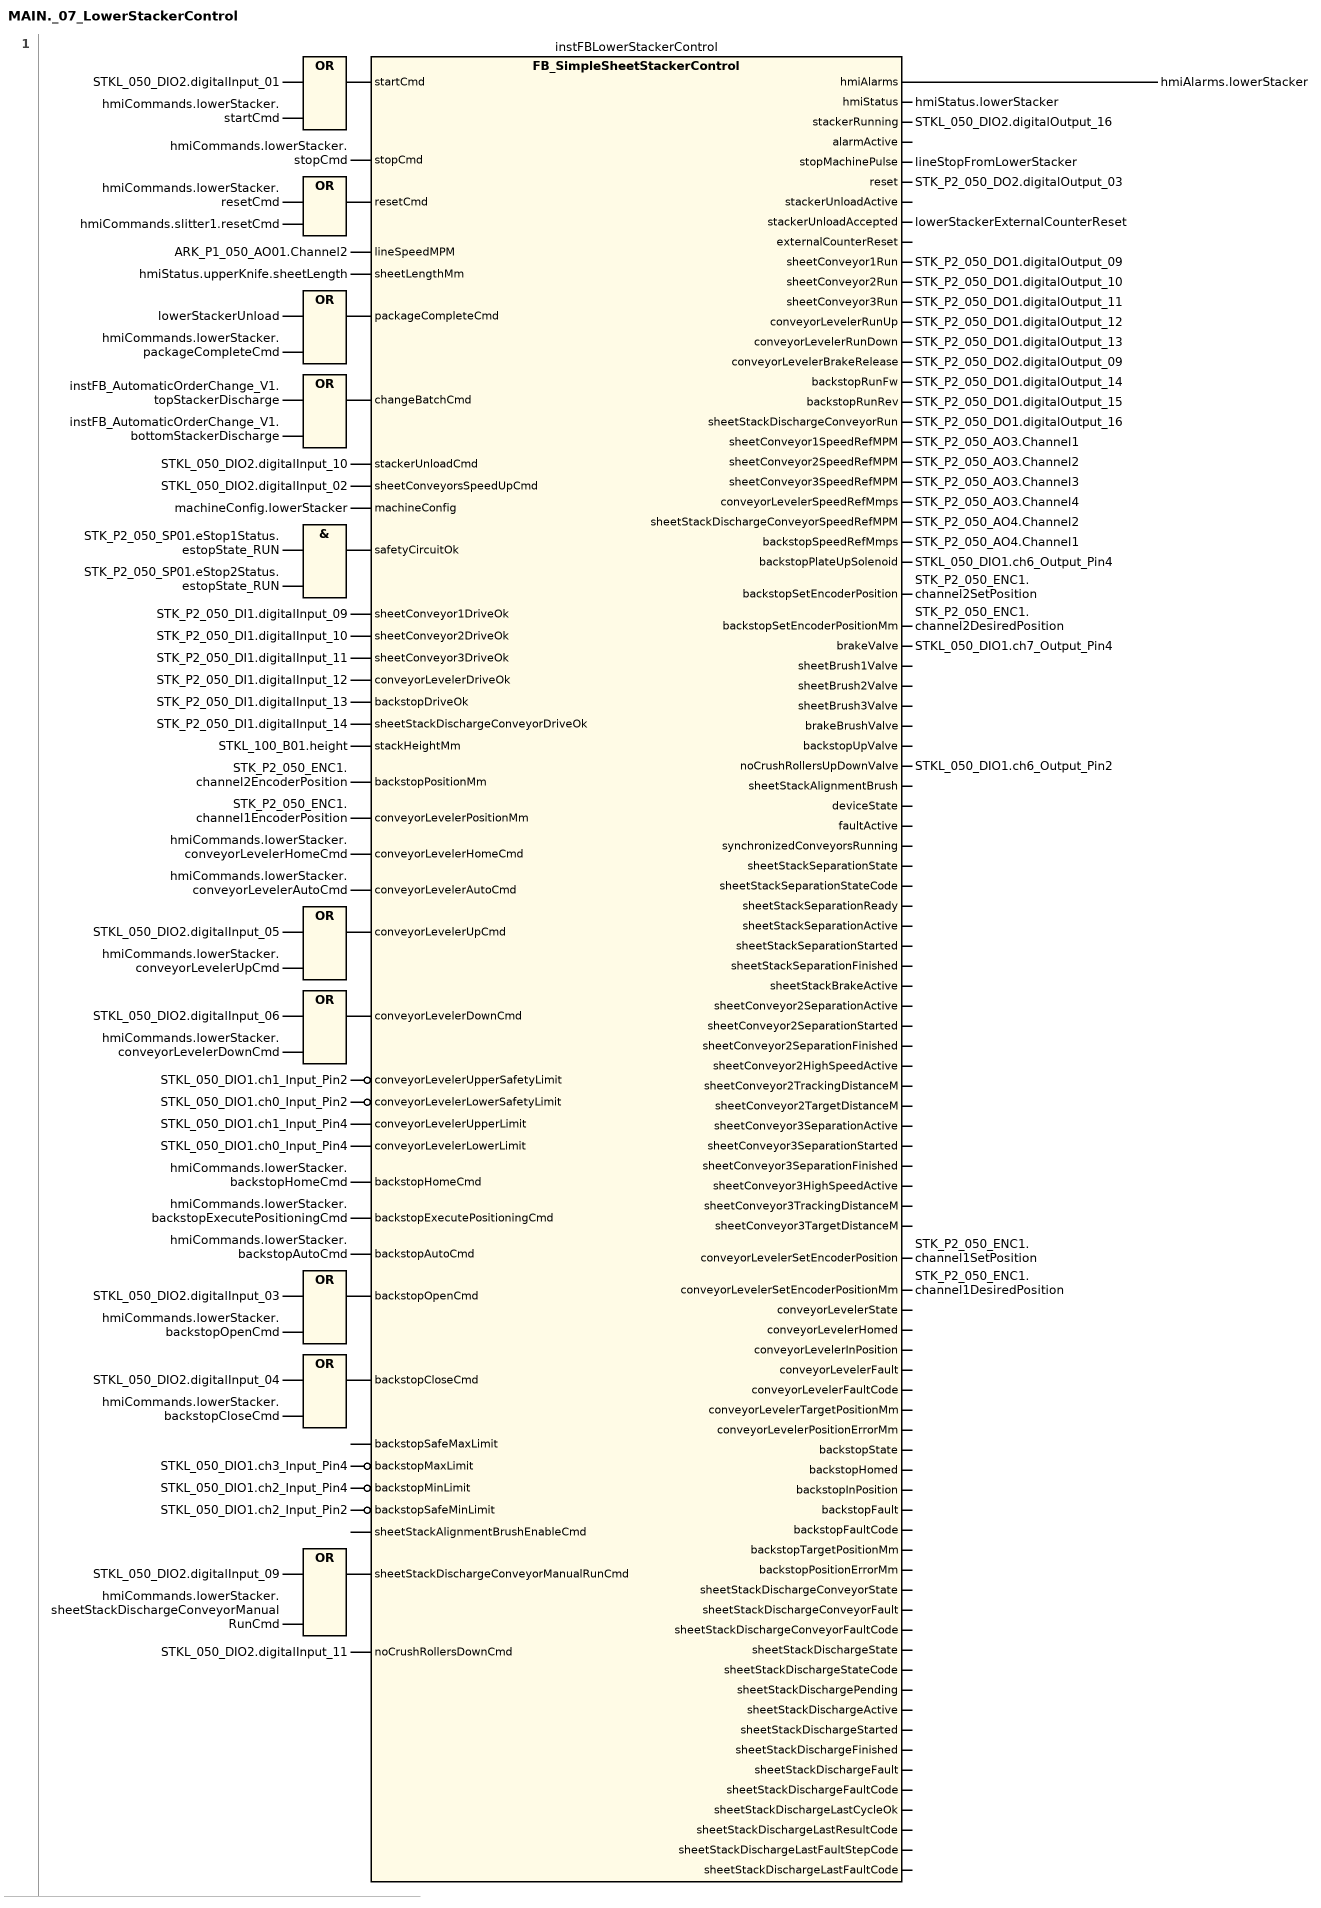
// NETWORK 1
instFBLowerStackerControl(
    startCmd := STKL_050_DIO2.digitalInput_01 OR hmiCommands.lowerStacker.startCmd,
    stopCmd := hmiCommands.lowerStacker.stopCmd,
    resetCmd := hmiCommands.lowerStacker.resetCmd OR hmiCommands.slitter1.resetCmd,
    lineSpeedMPM := ARK_P1_050_AO01.Channel2,
    sheetLengthMm := hmiStatus.upperKnife.sheetLength,
    packageCompleteCmd := lowerStackerUnload OR hmiCommands.lowerStacker.packageCompleteCmd,
    changeBatchCmd := instFB_AutomaticOrderChange_V1.topStackerDischarge OR instFB_AutomaticOrderChange_V1.bottomStackerDischarge,
    stackerUnloadCmd := STKL_050_DIO2.digitalInput_10,
    sheetConveyorsSpeedUpCmd := STKL_050_DIO2.digitalInput_02,
    machineConfig := machineConfig.lowerStacker,
    safetyCircuitOk := STK_P2_050_SP01.eStop1Status.estopState_RUN AND STK_P2_050_SP01.eStop2Status.estopState_RUN,
    sheetConveyor1DriveOk := STK_P2_050_DI1.digitalInput_09,
    sheetConveyor2DriveOk := STK_P2_050_DI1.digitalInput_10,
    sheetConveyor3DriveOk := STK_P2_050_DI1.digitalInput_11,
    conveyorLevelerDriveOk := STK_P2_050_DI1.digitalInput_12,
    backstopDriveOk := STK_P2_050_DI1.digitalInput_13,
    sheetStackDischargeConveyorDriveOk := STK_P2_050_DI1.digitalInput_14,
    stackHeightMm := STKL_100_B01.height,
    backstopPositionMm := STK_P2_050_ENC1.channel2EncoderPosition,
    conveyorLevelerPositionMm := STK_P2_050_ENC1.channel1EncoderPosition,
    conveyorLevelerHomeCmd := hmiCommands.lowerStacker.conveyorLevelerHomeCmd,
    conveyorLevelerAutoCmd := hmiCommands.lowerStacker.conveyorLevelerAutoCmd,
    conveyorLevelerUpCmd := STKL_050_DIO2.digitalInput_05 OR hmiCommands.lowerStacker.conveyorLevelerUpCmd,
    conveyorLevelerDownCmd := STKL_050_DIO2.digitalInput_06 OR hmiCommands.lowerStacker.conveyorLevelerDownCmd,
    conveyorLevelerUpperSafetyLimit := NOT STKL_050_DIO1.ch1_Input_Pin2,
    conveyorLevelerLowerSafetyLimit := NOT STKL_050_DIO1.ch0_Input_Pin2,
    conveyorLevelerUpperLimit := STKL_050_DIO1.ch1_Input_Pin4,
    conveyorLevelerLowerLimit := STKL_050_DIO1.ch0_Input_Pin4,
    backstopHomeCmd := hmiCommands.lowerStacker.backstopHomeCmd,
    backstopExecutePositioningCmd := hmiCommands.lowerStacker.backstopExecutePositioningCmd,
    backstopAutoCmd := hmiCommands.lowerStacker.backstopAutoCmd,
    backstopOpenCmd := STKL_050_DIO2.digitalInput_03 OR hmiCommands.lowerStacker.backstopOpenCmd,
    backstopCloseCmd := STKL_050_DIO2.digitalInput_04 OR hmiCommands.lowerStacker.backstopCloseCmd,
    backstopMaxLimit := NOT STKL_050_DIO1.ch3_Input_Pin4,
    backstopMinLimit := NOT STKL_050_DIO1.ch2_Input_Pin4,
    backstopSafeMinLimit := NOT STKL_050_DIO1.ch2_Input_Pin2,
    sheetStackDischargeConveyorManualRunCmd := STKL_050_DIO2.digitalInput_09 OR hmiCommands.lowerStacker.sheetStackDischargeConveyorManualRunCmd,
    noCrushRollersDownCmd := STKL_050_DIO2.digitalInput_11,
    hmiStatus => hmiStatus.lowerStacker,
    stackerRunning => STKL_050_DIO2.digitalOutput_16,
    stopMachinePulse => lineStopFromLowerStacker,
    reset => STK_P2_050_DO2.digitalOutput_03,
    stackerUnloadAccepted => lowerStackerExternalCounterReset,
    sheetConveyor1Run => STK_P2_050_DO1.digitalOutput_09,
    sheetConveyor2Run => STK_P2_050_DO1.digitalOutput_10,
    sheetConveyor3Run => STK_P2_050_DO1.digitalOutput_11,
    conveyorLevelerRunUp => STK_P2_050_DO1.digitalOutput_12,
    conveyorLevelerRunDown => STK_P2_050_DO1.digitalOutput_13,
    conveyorLevelerBrakeRelease => STK_P2_050_DO2.digitalOutput_09,
    backstopRunFw => STK_P2_050_DO1.digitalOutput_14,
    backstopRunRev => STK_P2_050_DO1.digitalOutput_15,
    sheetStackDischargeConveyorRun => STK_P2_050_DO1.digitalOutput_16,
    sheetConveyor1SpeedRefMPM => STK_P2_050_AO3.Channel1,
    sheetConveyor2SpeedRefMPM => STK_P2_050_AO3.Channel2,
    sheetConveyor3SpeedRefMPM => STK_P2_050_AO3.Channel3,
    conveyorLevelerSpeedRefMmps => STK_P2_050_AO3.Channel4,
    sheetStackDischargeConveyorSpeedRefMPM => STK_P2_050_AO4.Channel2,
    backstopSpeedRefMmps => STK_P2_050_AO4.Channel1,
    backstopPlateUpSolenoid => STKL_050_DIO1.ch6_Output_Pin4,
    backstopSetEncoderPosition => STK_P2_050_ENC1.channel2SetPosition,
    backstopSetEncoderPositionMm => STK_P2_050_ENC1.channel2DesiredPosition,
    brakeValve => STKL_050_DIO1.ch7_Output_Pin4,
    noCrushRollersUpDownValve => STKL_050_DIO1.ch6_Output_Pin2,
    conveyorLevelerSetEncoderPosition => STK_P2_050_ENC1.channel1SetPosition,
    conveyorLevelerSetEncoderPositionMm => STK_P2_050_ENC1.channel1DesiredPosition); // FB_SimpleSheetStackerControl
hmiAlarms.lowerStacker := instFBLowerStackerControl.hmiAlarms;

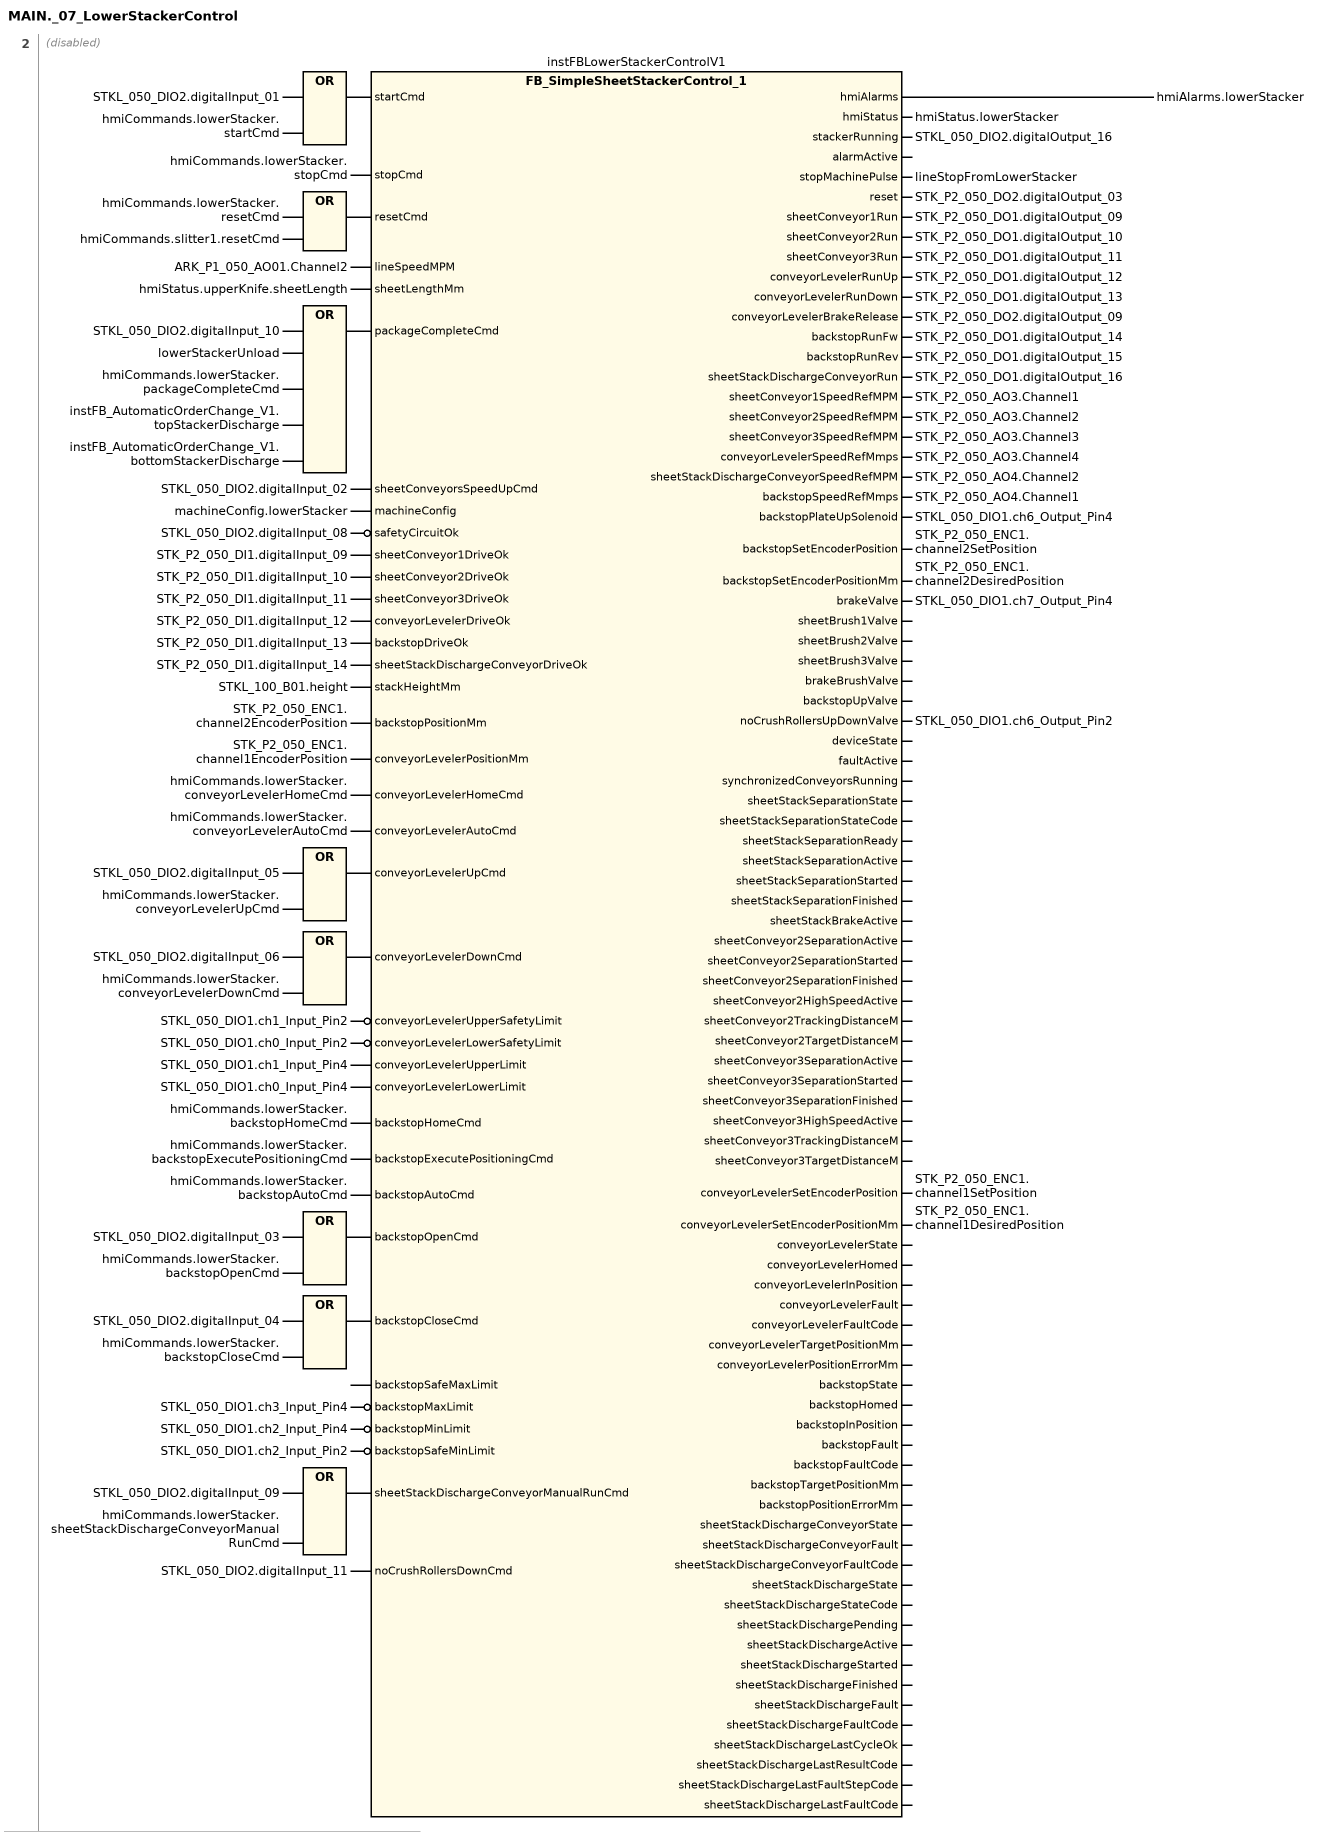
// NETWORK 2 (disabled)
// instFBLowerStackerControlV1(
//     startCmd := STKL_050_DIO2.digitalInput_01 OR hmiCommands.lowerStacker.startCmd,
//     stopCmd := hmiCommands.lowerStacker.stopCmd,
//     resetCmd := hmiCommands.lowerStacker.resetCmd OR hmiCommands.slitter1.resetCmd,
//     lineSpeedMPM := ARK_P1_050_AO01.Channel2,
//     sheetLengthMm := hmiStatus.upperKnife.sheetLength,
//     packageCompleteCmd := STKL_050_DIO2.digitalInput_10 OR lowerStackerUnload OR hmiCommands.lowerStacker.packageCompleteCmd OR instFB_AutomaticOrderChange_V1.topStackerDischarge OR instFB_AutomaticOrderChange_V1.bottomStackerDischarge,
//     sheetConveyorsSpeedUpCmd := STKL_050_DIO2.digitalInput_02,
//     machineConfig := machineConfig.lowerStacker,
//     safetyCircuitOk := NOT STKL_050_DIO2.digitalInput_08,
//     sheetConveyor1DriveOk := STK_P2_050_DI1.digitalInput_09,
//     sheetConveyor2DriveOk := STK_P2_050_DI1.digitalInput_10,
//     sheetConveyor3DriveOk := STK_P2_050_DI1.digitalInput_11,
//     conveyorLevelerDriveOk := STK_P2_050_DI1.digitalInput_12,
//     backstopDriveOk := STK_P2_050_DI1.digitalInput_13,
//     sheetStackDischargeConveyorDriveOk := STK_P2_050_DI1.digitalInput_14,
//     stackHeightMm := STKL_100_B01.height,
//     backstopPositionMm := STK_P2_050_ENC1.channel2EncoderPosition,
//     conveyorLevelerPositionMm := STK_P2_050_ENC1.channel1EncoderPosition,
//     conveyorLevelerHomeCmd := hmiCommands.lowerStacker.conveyorLevelerHomeCmd,
//     conveyorLevelerAutoCmd := hmiCommands.lowerStacker.conveyorLevelerAutoCmd,
//     conveyorLevelerUpCmd := STKL_050_DIO2.digitalInput_05 OR hmiCommands.lowerStacker.conveyorLevelerUpCmd,
//     conveyorLevelerDownCmd := STKL_050_DIO2.digitalInput_06 OR hmiCommands.lowerStacker.conveyorLevelerDownCmd,
//     conveyorLevelerUpperSafetyLimit := NOT STKL_050_DIO1.ch1_Input_Pin2,
//     conveyorLevelerLowerSafetyLimit := NOT STKL_050_DIO1.ch0_Input_Pin2,
//     conveyorLevelerUpperLimit := STKL_050_DIO1.ch1_Input_Pin4,
//     conveyorLevelerLowerLimit := STKL_050_DIO1.ch0_Input_Pin4,
//     backstopHomeCmd := hmiCommands.lowerStacker.backstopHomeCmd,
//     backstopExecutePositioningCmd := hmiCommands.lowerStacker.backstopExecutePositioningCmd,
//     backstopAutoCmd := hmiCommands.lowerStacker.backstopAutoCmd,
//     backstopOpenCmd := STKL_050_DIO2.digitalInput_03 OR hmiCommands.lowerStacker.backstopOpenCmd,
//     backstopCloseCmd := STKL_050_DIO2.digitalInput_04 OR hmiCommands.lowerStacker.backstopCloseCmd,
//     backstopMaxLimit := NOT STKL_050_DIO1.ch3_Input_Pin4,
//     backstopMinLimit := NOT STKL_050_DIO1.ch2_Input_Pin4,
//     backstopSafeMinLimit := NOT STKL_050_DIO1.ch2_Input_Pin2,
//     sheetStackDischargeConveyorManualRunCmd := STKL_050_DIO2.digitalInput_09 OR hmiCommands.lowerStacker.sheetStackDischargeConveyorManualRunCmd,
//     noCrushRollersDownCmd := STKL_050_DIO2.digitalInput_11,
//     hmiStatus => hmiStatus.lowerStacker,
//     stackerRunning => STKL_050_DIO2.digitalOutput_16,
//     stopMachinePulse => lineStopFromLowerStacker,
//     reset => STK_P2_050_DO2.digitalOutput_03,
//     sheetConveyor1Run => STK_P2_050_DO1.digitalOutput_09,
//     sheetConveyor2Run => STK_P2_050_DO1.digitalOutput_10,
//     sheetConveyor3Run => STK_P2_050_DO1.digitalOutput_11,
//     conveyorLevelerRunUp => STK_P2_050_DO1.digitalOutput_12,
//     conveyorLevelerRunDown => STK_P2_050_DO1.digitalOutput_13,
//     conveyorLevelerBrakeRelease => STK_P2_050_DO2.digitalOutput_09,
//     backstopRunFw => STK_P2_050_DO1.digitalOutput_14,
//     backstopRunRev => STK_P2_050_DO1.digitalOutput_15,
//     sheetStackDischargeConveyorRun => STK_P2_050_DO1.digitalOutput_16,
//     sheetConveyor1SpeedRefMPM => STK_P2_050_AO3.Channel1,
//     sheetConveyor2SpeedRefMPM => STK_P2_050_AO3.Channel2,
//     sheetConveyor3SpeedRefMPM => STK_P2_050_AO3.Channel3,
//     conveyorLevelerSpeedRefMmps => STK_P2_050_AO3.Channel4,
//     sheetStackDischargeConveyorSpeedRefMPM => STK_P2_050_AO4.Channel2,
//     backstopSpeedRefMmps => STK_P2_050_AO4.Channel1,
//     backstopPlateUpSolenoid => STKL_050_DIO1.ch6_Output_Pin4,
//     backstopSetEncoderPosition => STK_P2_050_ENC1.channel2SetPosition,
//     backstopSetEncoderPositionMm => STK_P2_050_ENC1.channel2DesiredPosition,
//     brakeValve => STKL_050_DIO1.ch7_Output_Pin4,
//     noCrushRollersUpDownValve => STKL_050_DIO1.ch6_Output_Pin2,
//     conveyorLevelerSetEncoderPosition => STK_P2_050_ENC1.channel1SetPosition,
//     conveyorLevelerSetEncoderPositionMm => STK_P2_050_ENC1.channel1DesiredPosition); // FB_SimpleSheetStackerControl_1
// hmiAlarms.lowerStacker := instFBLowerStackerControlV1.hmiAlarms;
END_METHOD

METHOD _08_UpperStackerControl
VAR_INPUT
END_VAR
//STKU_050_DIO2.digitalInput_12 Material no backstop
VAR

END_VAR
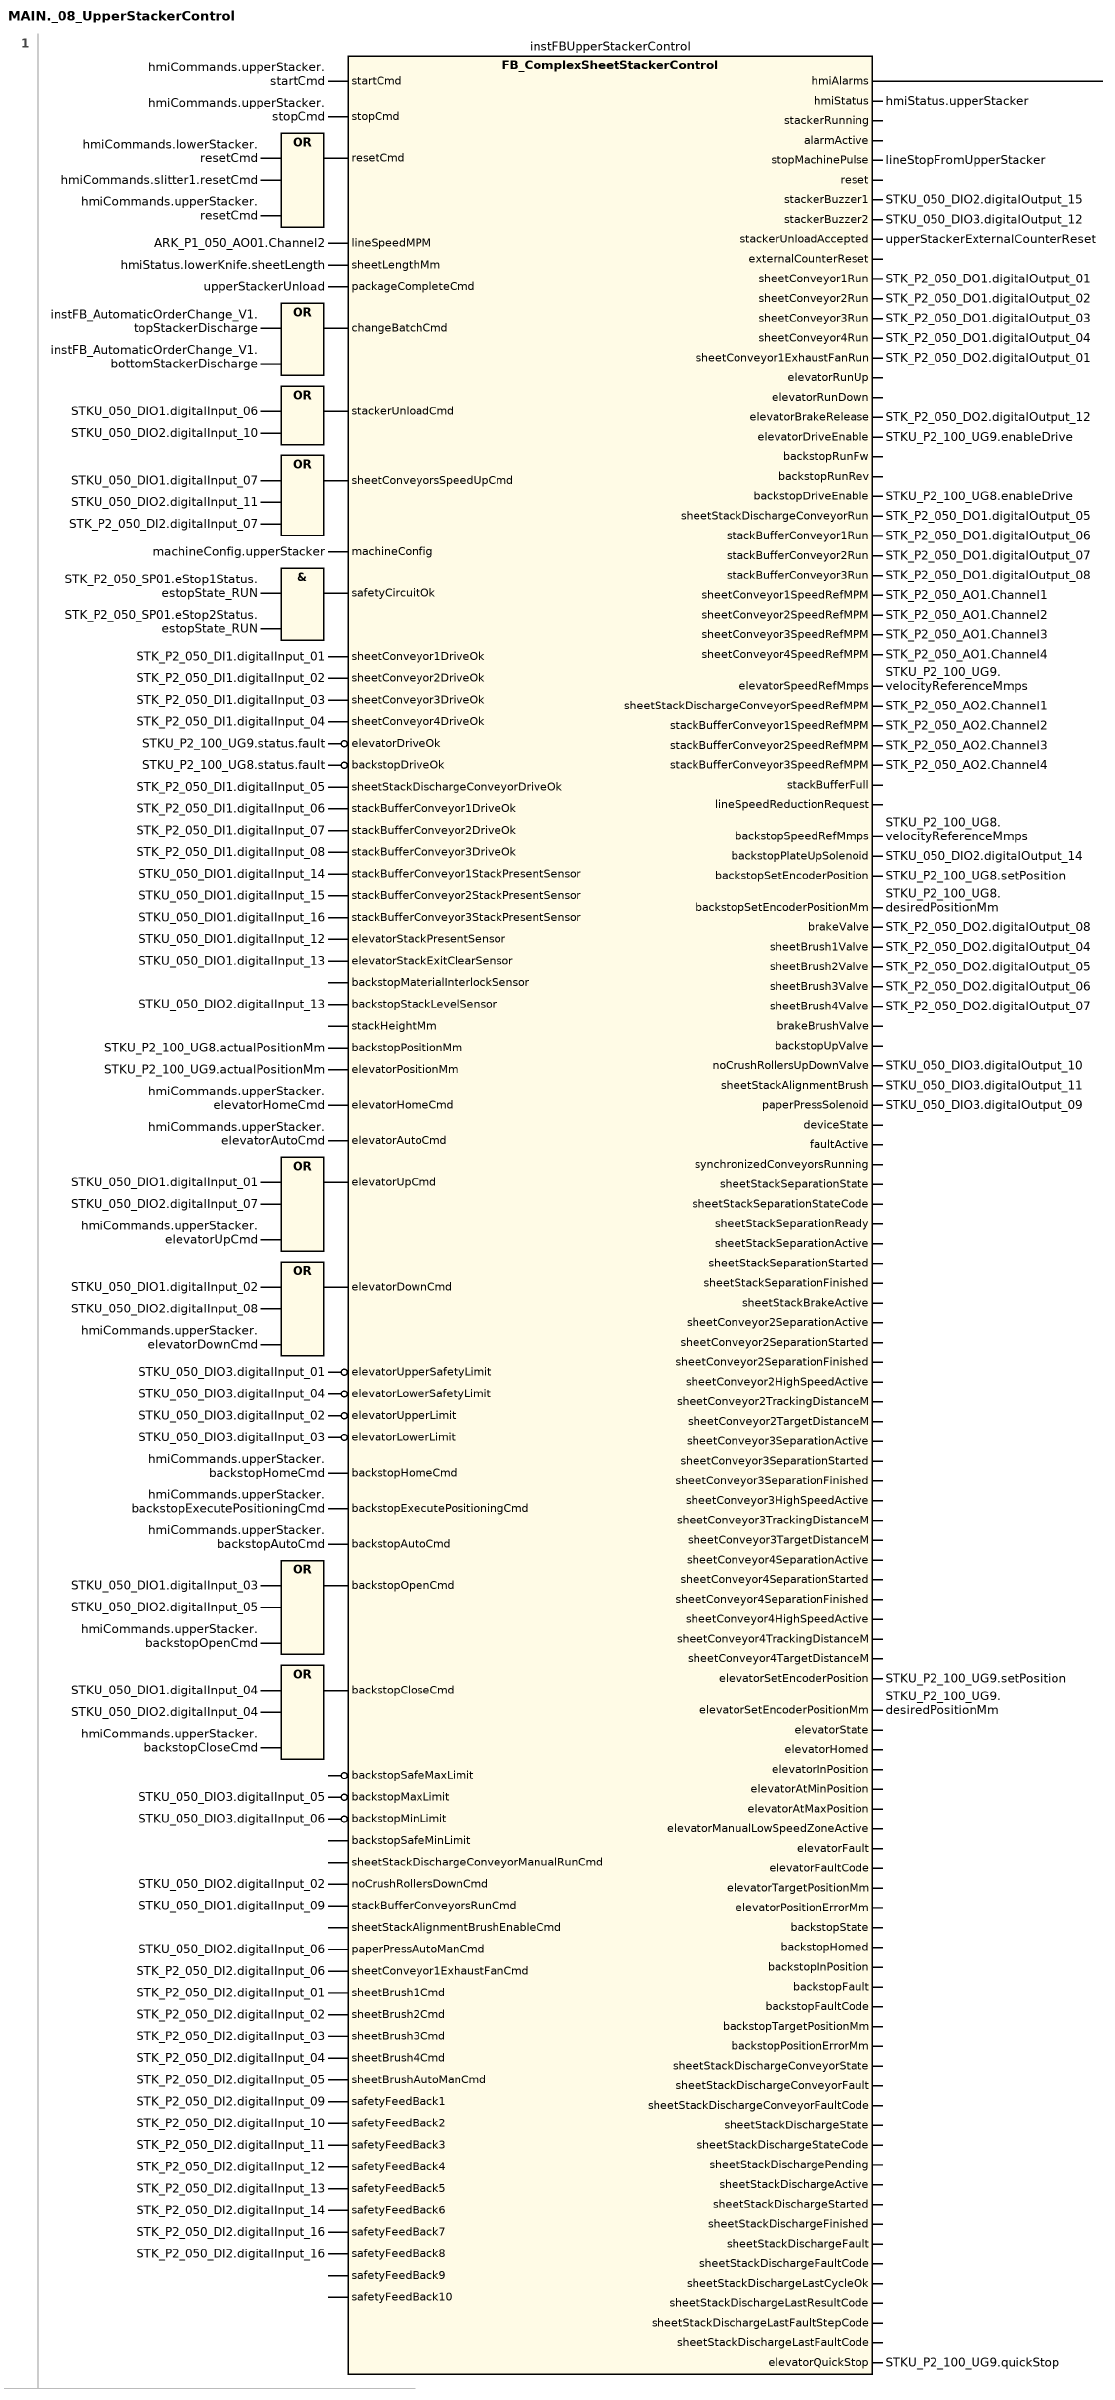
// NETWORK 1
instFBUpperStackerControl(
    startCmd := hmiCommands.upperStacker.startCmd,
    stopCmd := hmiCommands.upperStacker.stopCmd,
    resetCmd := hmiCommands.lowerStacker.resetCmd OR hmiCommands.slitter1.resetCmd OR hmiCommands.upperStacker.resetCmd,
    lineSpeedMPM := ARK_P1_050_AO01.Channel2,
    sheetLengthMm := hmiStatus.lowerKnife.sheetLength,
    packageCompleteCmd := upperStackerUnload,
    changeBatchCmd := instFB_AutomaticOrderChange_V1.topStackerDischarge OR instFB_AutomaticOrderChange_V1.bottomStackerDischarge,
    stackerUnloadCmd := STKU_050_DIO1.digitalInput_06 OR STKU_050_DIO2.digitalInput_10,
    sheetConveyorsSpeedUpCmd := STKU_050_DIO1.digitalInput_07 OR STKU_050_DIO2.digitalInput_11 OR STK_P2_050_DI2.digitalInput_07,
    machineConfig := machineConfig.upperStacker,
    safetyCircuitOk := STK_P2_050_SP01.eStop1Status.estopState_RUN AND STK_P2_050_SP01.eStop2Status.estopState_RUN,
    sheetConveyor1DriveOk := STK_P2_050_DI1.digitalInput_01,
    sheetConveyor2DriveOk := STK_P2_050_DI1.digitalInput_02,
    sheetConveyor3DriveOk := STK_P2_050_DI1.digitalInput_03,
    sheetConveyor4DriveOk := STK_P2_050_DI1.digitalInput_04,
    elevatorDriveOk := NOT STKU_P2_100_UG9.status.fault,
    backstopDriveOk := NOT STKU_P2_100_UG8.status.fault,
    sheetStackDischargeConveyorDriveOk := STK_P2_050_DI1.digitalInput_05,
    stackBufferConveyor1DriveOk := STK_P2_050_DI1.digitalInput_06,
    stackBufferConveyor2DriveOk := STK_P2_050_DI1.digitalInput_07,
    stackBufferConveyor3DriveOk := STK_P2_050_DI1.digitalInput_08,
    stackBufferConveyor1StackPresentSensor := STKU_050_DIO1.digitalInput_14,
    stackBufferConveyor2StackPresentSensor := STKU_050_DIO1.digitalInput_15,
    stackBufferConveyor3StackPresentSensor := STKU_050_DIO1.digitalInput_16,
    elevatorStackPresentSensor := STKU_050_DIO1.digitalInput_12,
    elevatorStackExitClearSensor := STKU_050_DIO1.digitalInput_13,
    backstopStackLevelSensor := STKU_050_DIO2.digitalInput_13,
    backstopPositionMm := STKU_P2_100_UG8.actualPositionMm,
    elevatorPositionMm := STKU_P2_100_UG9.actualPositionMm,
    elevatorHomeCmd := hmiCommands.upperStacker.elevatorHomeCmd,
    elevatorAutoCmd := hmiCommands.upperStacker.elevatorAutoCmd,
    elevatorUpCmd := STKU_050_DIO1.digitalInput_01 OR STKU_050_DIO2.digitalInput_07 OR hmiCommands.upperStacker.elevatorUpCmd,
    elevatorDownCmd := STKU_050_DIO1.digitalInput_02 OR STKU_050_DIO2.digitalInput_08 OR hmiCommands.upperStacker.elevatorDownCmd,
    elevatorUpperSafetyLimit := NOT STKU_050_DIO3.digitalInput_01,
    elevatorLowerSafetyLimit := NOT STKU_050_DIO3.digitalInput_04,
    elevatorUpperLimit := NOT STKU_050_DIO3.digitalInput_02,
    elevatorLowerLimit := NOT STKU_050_DIO3.digitalInput_03,
    backstopHomeCmd := hmiCommands.upperStacker.backstopHomeCmd,
    backstopExecutePositioningCmd := hmiCommands.upperStacker.backstopExecutePositioningCmd,
    backstopAutoCmd := hmiCommands.upperStacker.backstopAutoCmd,
    backstopOpenCmd := STKU_050_DIO1.digitalInput_03 OR STKU_050_DIO2.digitalInput_05 OR hmiCommands.upperStacker.backstopOpenCmd,
    backstopCloseCmd := STKU_050_DIO1.digitalInput_04 OR STKU_050_DIO2.digitalInput_04 OR hmiCommands.upperStacker.backstopCloseCmd,
    backstopMaxLimit := NOT STKU_050_DIO3.digitalInput_05,
    backstopMinLimit := NOT STKU_050_DIO3.digitalInput_06,
    noCrushRollersDownCmd := STKU_050_DIO2.digitalInput_02,
    stackBufferConveyorsRunCmd := STKU_050_DIO1.digitalInput_09,
    paperPressAutoManCmd := STKU_050_DIO2.digitalInput_06,
    sheetConveyor1ExhaustFanCmd := STK_P2_050_DI2.digitalInput_06,
    sheetBrush1Cmd := STK_P2_050_DI2.digitalInput_01,
    sheetBrush2Cmd := STK_P2_050_DI2.digitalInput_02,
    sheetBrush3Cmd := STK_P2_050_DI2.digitalInput_03,
    sheetBrush4Cmd := STK_P2_050_DI2.digitalInput_04,
    sheetBrushAutoManCmd := STK_P2_050_DI2.digitalInput_05,
    safetyFeedBack1 := STK_P2_050_DI2.digitalInput_09,
    safetyFeedBack2 := STK_P2_050_DI2.digitalInput_10,
    safetyFeedBack3 := STK_P2_050_DI2.digitalInput_11,
    safetyFeedBack4 := STK_P2_050_DI2.digitalInput_12,
    safetyFeedBack5 := STK_P2_050_DI2.digitalInput_13,
    safetyFeedBack6 := STK_P2_050_DI2.digitalInput_14,
    safetyFeedBack7 := STK_P2_050_DI2.digitalInput_16,
    safetyFeedBack8 := STK_P2_050_DI2.digitalInput_16,
    hmiStatus => hmiStatus.upperStacker,
    stopMachinePulse => lineStopFromUpperStacker,
    stackerBuzzer1 => STKU_050_DIO2.digitalOutput_15,
    stackerBuzzer2 => STKU_050_DIO3.digitalOutput_12,
    stackerUnloadAccepted => upperStackerExternalCounterReset,
    sheetConveyor1Run => STK_P2_050_DO1.digitalOutput_01,
    sheetConveyor2Run => STK_P2_050_DO1.digitalOutput_02,
    sheetConveyor3Run => STK_P2_050_DO1.digitalOutput_03,
    sheetConveyor4Run => STK_P2_050_DO1.digitalOutput_04,
    sheetConveyor1ExhaustFanRun => STK_P2_050_DO2.digitalOutput_01,
    elevatorBrakeRelease => STK_P2_050_DO2.digitalOutput_12,
    elevatorDriveEnable => STKU_P2_100_UG9.enableDrive,
    backstopDriveEnable => STKU_P2_100_UG8.enableDrive,
    sheetStackDischargeConveyorRun => STK_P2_050_DO1.digitalOutput_05,
    stackBufferConveyor1Run => STK_P2_050_DO1.digitalOutput_06,
    stackBufferConveyor2Run => STK_P2_050_DO1.digitalOutput_07,
    stackBufferConveyor3Run => STK_P2_050_DO1.digitalOutput_08,
    sheetConveyor1SpeedRefMPM => STK_P2_050_AO1.Channel1,
    sheetConveyor2SpeedRefMPM => STK_P2_050_AO1.Channel2,
    sheetConveyor3SpeedRefMPM => STK_P2_050_AO1.Channel3,
    sheetConveyor4SpeedRefMPM => STK_P2_050_AO1.Channel4,
    elevatorSpeedRefMmps => STKU_P2_100_UG9.velocityReferenceMmps,
    sheetStackDischargeConveyorSpeedRefMPM => STK_P2_050_AO2.Channel1,
    stackBufferConveyor1SpeedRefMPM => STK_P2_050_AO2.Channel2,
    stackBufferConveyor2SpeedRefMPM => STK_P2_050_AO2.Channel3,
    stackBufferConveyor3SpeedRefMPM => STK_P2_050_AO2.Channel4,
    backstopSpeedRefMmps => STKU_P2_100_UG8.velocityReferenceMmps,
    backstopPlateUpSolenoid => STKU_050_DIO2.digitalOutput_14,
    backstopSetEncoderPosition => STKU_P2_100_UG8.setPosition,
    backstopSetEncoderPositionMm => STKU_P2_100_UG8.desiredPositionMm,
    brakeValve => STK_P2_050_DO2.digitalOutput_08,
    sheetBrush1Valve => STK_P2_050_DO2.digitalOutput_04,
    sheetBrush2Valve => STK_P2_050_DO2.digitalOutput_05,
    sheetBrush3Valve => STK_P2_050_DO2.digitalOutput_06,
    sheetBrush4Valve => STK_P2_050_DO2.digitalOutput_07,
    noCrushRollersUpDownValve => STKU_050_DIO3.digitalOutput_10,
    sheetStackAlignmentBrush => STKU_050_DIO3.digitalOutput_11,
    paperPressSolenoid => STKU_050_DIO3.digitalOutput_09,
    elevatorSetEncoderPosition => STKU_P2_100_UG9.setPosition,
    elevatorSetEncoderPositionMm => STKU_P2_100_UG9.desiredPositionMm,
    elevatorQuickStop => STKU_P2_100_UG9.quickStop); // FB_ComplexSheetStackerControl
END_METHOD

ACTION ACT_Slitter1Control:
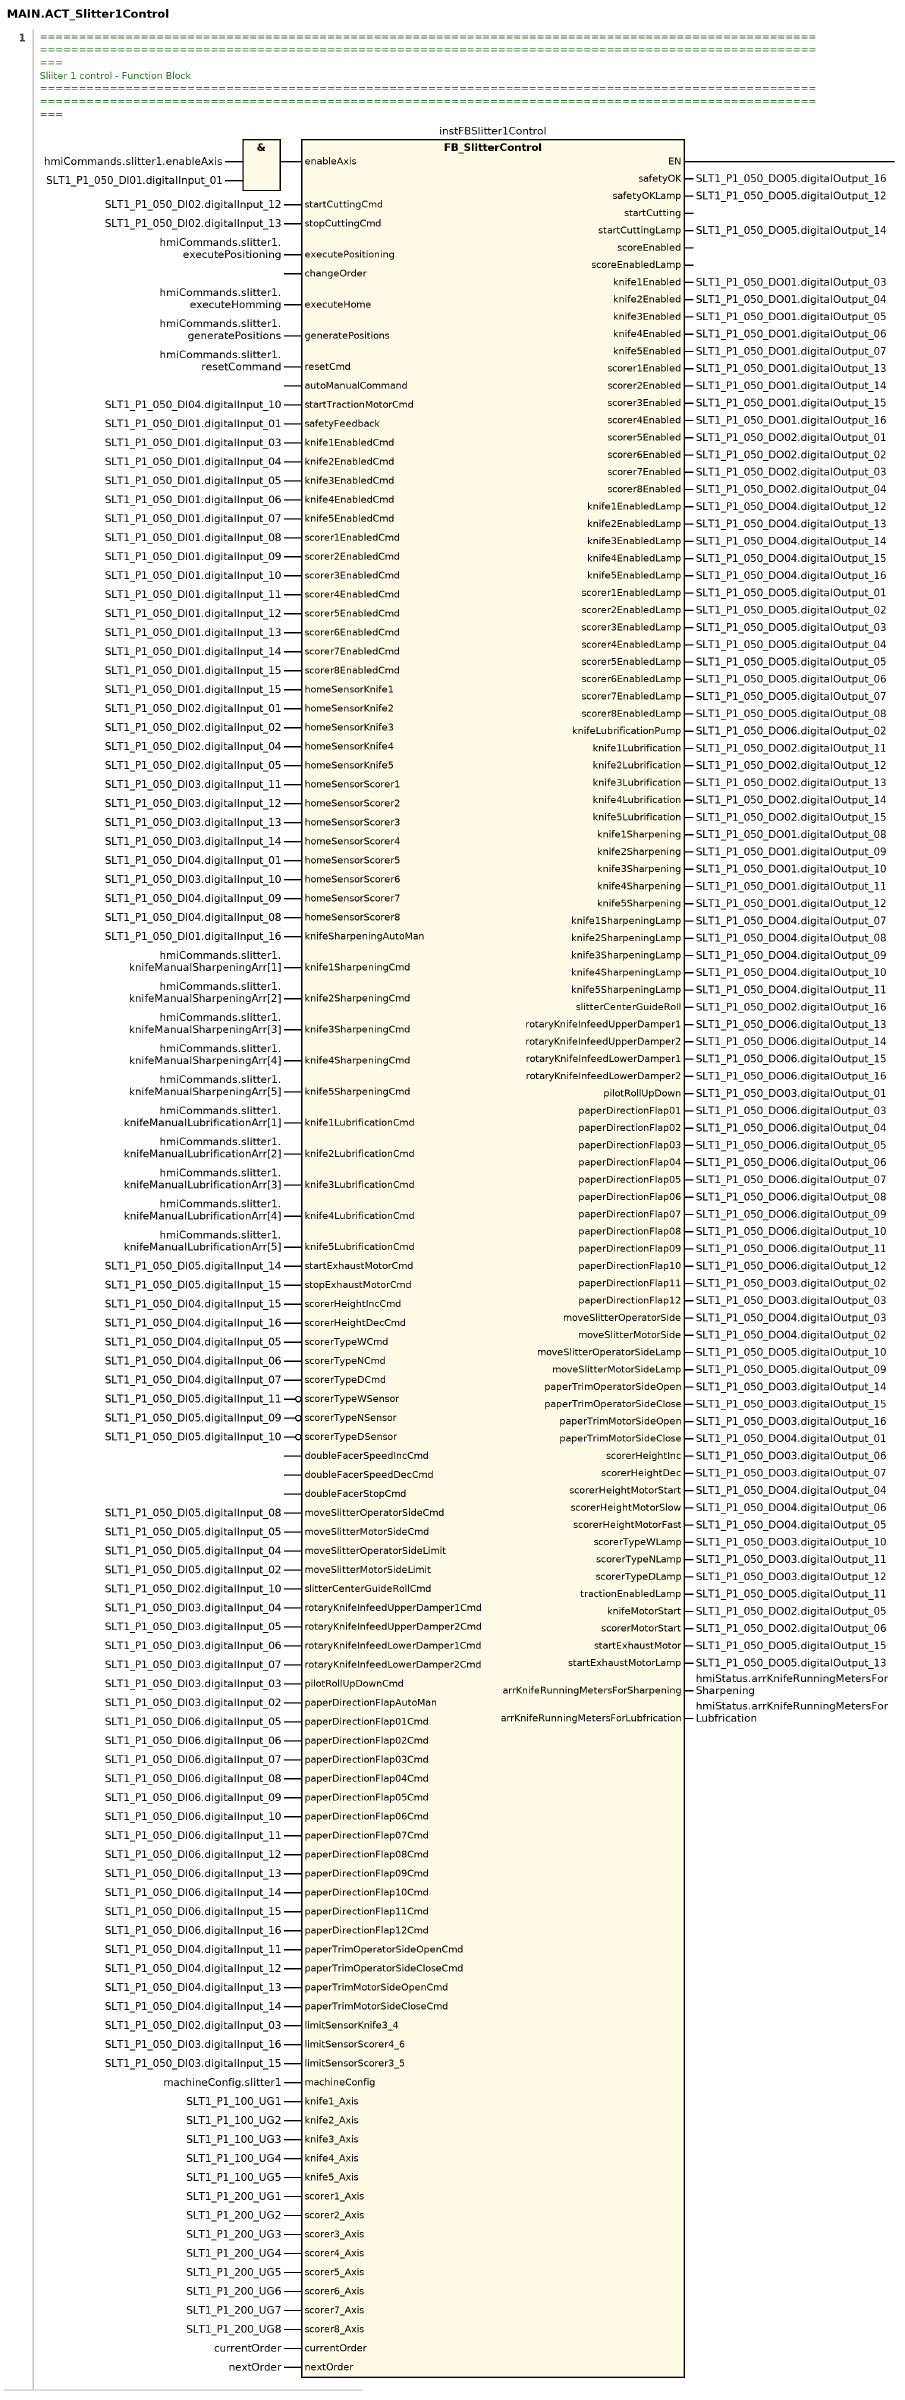
// NETWORK 1
// 					===========================================================================================================================================================================================================
//
// Sliiter 1 control - Function Block
//
// ===========================================================================================================================================================================================================
//
instFBSlitter1Control(
    enableAxis := hmiCommands.slitter1.enableAxis AND SLT1_P1_050_DI01.digitalInput_01,
    startCuttingCmd := SLT1_P1_050_DI02.digitalInput_12,
    stopCuttingCmd := SLT1_P1_050_DI02.digitalInput_13,
    executePositioning := hmiCommands.slitter1.executePositioning,
    executeHome := hmiCommands.slitter1.executeHomming,
    generatePositions := hmiCommands.slitter1.generatePositions,
    resetCmd := hmiCommands.slitter1.resetCommand,
    startTractionMotorCmd := SLT1_P1_050_DI04.digitalInput_10,
    safetyFeedback := SLT1_P1_050_DI01.digitalInput_01,
    knife1EnabledCmd := SLT1_P1_050_DI01.digitalInput_03,
    knife2EnabledCmd := SLT1_P1_050_DI01.digitalInput_04,
    knife3EnabledCmd := SLT1_P1_050_DI01.digitalInput_05,
    knife4EnabledCmd := SLT1_P1_050_DI01.digitalInput_06,
    knife5EnabledCmd := SLT1_P1_050_DI01.digitalInput_07,
    scorer1EnabledCmd := SLT1_P1_050_DI01.digitalInput_08,
    scorer2EnabledCmd := SLT1_P1_050_DI01.digitalInput_09,
    scorer3EnabledCmd := SLT1_P1_050_DI01.digitalInput_10,
    scorer4EnabledCmd := SLT1_P1_050_DI01.digitalInput_11,
    scorer5EnabledCmd := SLT1_P1_050_DI01.digitalInput_12,
    scorer6EnabledCmd := SLT1_P1_050_DI01.digitalInput_13,
    scorer7EnabledCmd := SLT1_P1_050_DI01.digitalInput_14,
    scorer8EnabledCmd := SLT1_P1_050_DI01.digitalInput_15,
    homeSensorKnife1 := SLT1_P1_050_DI01.digitalInput_15,
    homeSensorKnife2 := SLT1_P1_050_DI02.digitalInput_01,
    homeSensorKnife3 := SLT1_P1_050_DI02.digitalInput_02,
    homeSensorKnife4 := SLT1_P1_050_DI02.digitalInput_04,
    homeSensorKnife5 := SLT1_P1_050_DI02.digitalInput_05,
    homeSensorScorer1 := SLT1_P1_050_DI03.digitalInput_11,
    homeSensorScorer2 := SLT1_P1_050_DI03.digitalInput_12,
    homeSensorScorer3 := SLT1_P1_050_DI03.digitalInput_13,
    homeSensorScorer4 := SLT1_P1_050_DI03.digitalInput_14,
    homeSensorScorer5 := SLT1_P1_050_DI04.digitalInput_01,
    homeSensorScorer6 := SLT1_P1_050_DI03.digitalInput_10,
    homeSensorScorer7 := SLT1_P1_050_DI04.digitalInput_09,
    homeSensorScorer8 := SLT1_P1_050_DI04.digitalInput_08,
    knifeSharpeningAutoMan := SLT1_P1_050_DI01.digitalInput_16,
    knife1SharpeningCmd := hmiCommands.slitter1.knifeManualSharpeningArr[1],
    knife2SharpeningCmd := hmiCommands.slitter1.knifeManualSharpeningArr[2],
    knife3SharpeningCmd := hmiCommands.slitter1.knifeManualSharpeningArr[3],
    knife4SharpeningCmd := hmiCommands.slitter1.knifeManualSharpeningArr[4],
    knife5SharpeningCmd := hmiCommands.slitter1.knifeManualSharpeningArr[5],
    knife1LubrificationCmd := hmiCommands.slitter1.knifeManualLubrificationArr[1],
    knife2LubrificationCmd := hmiCommands.slitter1.knifeManualLubrificationArr[2],
    knife3LubrificationCmd := hmiCommands.slitter1.knifeManualLubrificationArr[3],
    knife4LubrificationCmd := hmiCommands.slitter1.knifeManualLubrificationArr[4],
    knife5LubrificationCmd := hmiCommands.slitter1.knifeManualLubrificationArr[5],
    startExhaustMotorCmd := SLT1_P1_050_DI05.digitalInput_14,
    stopExhaustMotorCmd := SLT1_P1_050_DI05.digitalInput_15,
    scorerHeightIncCmd := SLT1_P1_050_DI04.digitalInput_15,
    scorerHeightDecCmd := SLT1_P1_050_DI04.digitalInput_16,
    scorerTypeWCmd := SLT1_P1_050_DI04.digitalInput_05,
    scorerTypeNCmd := SLT1_P1_050_DI04.digitalInput_06,
    scorerTypeDCmd := SLT1_P1_050_DI04.digitalInput_07,
    scorerTypeWSensor := NOT SLT1_P1_050_DI05.digitalInput_11,
    scorerTypeNSensor := NOT SLT1_P1_050_DI05.digitalInput_09,
    scorerTypeDSensor := NOT SLT1_P1_050_DI05.digitalInput_10,
    moveSlitterOperatorSideCmd := SLT1_P1_050_DI05.digitalInput_08,
    moveSlitterMotorSideCmd := SLT1_P1_050_DI05.digitalInput_05,
    moveSlitterOperatorSideLimit := SLT1_P1_050_DI05.digitalInput_04,
    moveSlitterMotorSideLimit := SLT1_P1_050_DI05.digitalInput_02,
    slitterCenterGuideRollCmd := SLT1_P1_050_DI02.digitalInput_10,
    rotaryKnifeInfeedUpperDamper1Cmd := SLT1_P1_050_DI03.digitalInput_04,
    rotaryKnifeInfeedUpperDamper2Cmd := SLT1_P1_050_DI03.digitalInput_05,
    rotaryKnifeInfeedLowerDamper1Cmd := SLT1_P1_050_DI03.digitalInput_06,
    rotaryKnifeInfeedLowerDamper2Cmd := SLT1_P1_050_DI03.digitalInput_07,
    pilotRollUpDownCmd := SLT1_P1_050_DI03.digitalInput_03,
    paperDirectionFlapAutoMan := SLT1_P1_050_DI03.digitalInput_02,
    paperDirectionFlap01Cmd := SLT1_P1_050_DI06.digitalInput_05,
    paperDirectionFlap02Cmd := SLT1_P1_050_DI06.digitalInput_06,
    paperDirectionFlap03Cmd := SLT1_P1_050_DI06.digitalInput_07,
    paperDirectionFlap04Cmd := SLT1_P1_050_DI06.digitalInput_08,
    paperDirectionFlap05Cmd := SLT1_P1_050_DI06.digitalInput_09,
    paperDirectionFlap06Cmd := SLT1_P1_050_DI06.digitalInput_10,
    paperDirectionFlap07Cmd := SLT1_P1_050_DI06.digitalInput_11,
    paperDirectionFlap08Cmd := SLT1_P1_050_DI06.digitalInput_12,
    paperDirectionFlap09Cmd := SLT1_P1_050_DI06.digitalInput_13,
    paperDirectionFlap10Cmd := SLT1_P1_050_DI06.digitalInput_14,
    paperDirectionFlap11Cmd := SLT1_P1_050_DI06.digitalInput_15,
    paperDirectionFlap12Cmd := SLT1_P1_050_DI06.digitalInput_16,
    paperTrimOperatorSideOpenCmd := SLT1_P1_050_DI04.digitalInput_11,
    paperTrimOperatorSideCloseCmd := SLT1_P1_050_DI04.digitalInput_12,
    paperTrimMotorSideOpenCmd := SLT1_P1_050_DI04.digitalInput_13,
    paperTrimMotorSideCloseCmd := SLT1_P1_050_DI04.digitalInput_14,
    limitSensorKnife3_4 := SLT1_P1_050_DI02.digitalInput_03,
    limitSensorScorer4_6 := SLT1_P1_050_DI03.digitalInput_16,
    limitSensorScorer3_5 := SLT1_P1_050_DI03.digitalInput_15,
    machineConfig := machineConfig.slitter1,
    knife1_Axis := SLT1_P1_100_UG1,
    knife2_Axis := SLT1_P1_100_UG2,
    knife3_Axis := SLT1_P1_100_UG3,
    knife4_Axis := SLT1_P1_100_UG4,
    knife5_Axis := SLT1_P1_100_UG5,
    scorer1_Axis := SLT1_P1_200_UG1,
    scorer2_Axis := SLT1_P1_200_UG2,
    scorer3_Axis := SLT1_P1_200_UG3,
    scorer4_Axis := SLT1_P1_200_UG4,
    scorer5_Axis := SLT1_P1_200_UG5,
    scorer6_Axis := SLT1_P1_200_UG6,
    scorer7_Axis := SLT1_P1_200_UG7,
    scorer8_Axis := SLT1_P1_200_UG8,
    currentOrder := currentOrder,
    nextOrder := nextOrder,
    safetyOK => SLT1_P1_050_DO05.digitalOutput_16,
    safetyOKLamp => SLT1_P1_050_DO05.digitalOutput_12,
    startCuttingLamp => SLT1_P1_050_DO05.digitalOutput_14,
    knife1Enabled => SLT1_P1_050_DO01.digitalOutput_03,
    knife2Enabled => SLT1_P1_050_DO01.digitalOutput_04,
    knife3Enabled => SLT1_P1_050_DO01.digitalOutput_05,
    knife4Enabled => SLT1_P1_050_DO01.digitalOutput_06,
    knife5Enabled => SLT1_P1_050_DO01.digitalOutput_07,
    scorer1Enabled => SLT1_P1_050_DO01.digitalOutput_13,
    scorer2Enabled => SLT1_P1_050_DO01.digitalOutput_14,
    scorer3Enabled => SLT1_P1_050_DO01.digitalOutput_15,
    scorer4Enabled => SLT1_P1_050_DO01.digitalOutput_16,
    scorer5Enabled => SLT1_P1_050_DO02.digitalOutput_01,
    scorer6Enabled => SLT1_P1_050_DO02.digitalOutput_02,
    scorer7Enabled => SLT1_P1_050_DO02.digitalOutput_03,
    scorer8Enabled => SLT1_P1_050_DO02.digitalOutput_04,
    knife1EnabledLamp => SLT1_P1_050_DO04.digitalOutput_12,
    knife2EnabledLamp => SLT1_P1_050_DO04.digitalOutput_13,
    knife3EnabledLamp => SLT1_P1_050_DO04.digitalOutput_14,
    knife4EnabledLamp => SLT1_P1_050_DO04.digitalOutput_15,
    knife5EnabledLamp => SLT1_P1_050_DO04.digitalOutput_16,
    scorer1EnabledLamp => SLT1_P1_050_DO05.digitalOutput_01,
    scorer2EnabledLamp => SLT1_P1_050_DO05.digitalOutput_02,
    scorer3EnabledLamp => SLT1_P1_050_DO05.digitalOutput_03,
    scorer4EnabledLamp => SLT1_P1_050_DO05.digitalOutput_04,
    scorer5EnabledLamp => SLT1_P1_050_DO05.digitalOutput_05,
    scorer6EnabledLamp => SLT1_P1_050_DO05.digitalOutput_06,
    scorer7EnabledLamp => SLT1_P1_050_DO05.digitalOutput_07,
    scorer8EnabledLamp => SLT1_P1_050_DO05.digitalOutput_08,
    knifeLubrificationPump => SLT1_P1_050_DO06.digitalOutput_02,
    knife1Lubrification => SLT1_P1_050_DO02.digitalOutput_11,
    knife2Lubrification => SLT1_P1_050_DO02.digitalOutput_12,
    knife3Lubrification => SLT1_P1_050_DO02.digitalOutput_13,
    knife4Lubrification => SLT1_P1_050_DO02.digitalOutput_14,
    knife5Lubrification => SLT1_P1_050_DO02.digitalOutput_15,
    knife1Sharpening => SLT1_P1_050_DO01.digitalOutput_08,
    knife2Sharpening => SLT1_P1_050_DO01.digitalOutput_09,
    knife3Sharpening => SLT1_P1_050_DO01.digitalOutput_10,
    knife4Sharpening => SLT1_P1_050_DO01.digitalOutput_11,
    knife5Sharpening => SLT1_P1_050_DO01.digitalOutput_12,
    knife1SharpeningLamp => SLT1_P1_050_DO04.digitalOutput_07,
    knife2SharpeningLamp => SLT1_P1_050_DO04.digitalOutput_08,
    knife3SharpeningLamp => SLT1_P1_050_DO04.digitalOutput_09,
    knife4SharpeningLamp => SLT1_P1_050_DO04.digitalOutput_10,
    knife5SharpeningLamp => SLT1_P1_050_DO04.digitalOutput_11,
    slitterCenterGuideRoll => SLT1_P1_050_DO02.digitalOutput_16,
    rotaryKnifeInfeedUpperDamper1 => SLT1_P1_050_DO06.digitalOutput_13,
    rotaryKnifeInfeedUpperDamper2 => SLT1_P1_050_DO06.digitalOutput_14,
    rotaryKnifeInfeedLowerDamper1 => SLT1_P1_050_DO06.digitalOutput_15,
    rotaryKnifeInfeedLowerDamper2 => SLT1_P1_050_DO06.digitalOutput_16,
    pilotRollUpDown => SLT1_P1_050_DO03.digitalOutput_01,
    paperDirectionFlap01 => SLT1_P1_050_DO06.digitalOutput_03,
    paperDirectionFlap02 => SLT1_P1_050_DO06.digitalOutput_04,
    paperDirectionFlap03 => SLT1_P1_050_DO06.digitalOutput_05,
    paperDirectionFlap04 => SLT1_P1_050_DO06.digitalOutput_06,
    paperDirectionFlap05 => SLT1_P1_050_DO06.digitalOutput_07,
    paperDirectionFlap06 => SLT1_P1_050_DO06.digitalOutput_08,
    paperDirectionFlap07 => SLT1_P1_050_DO06.digitalOutput_09,
    paperDirectionFlap08 => SLT1_P1_050_DO06.digitalOutput_10,
    paperDirectionFlap09 => SLT1_P1_050_DO06.digitalOutput_11,
    paperDirectionFlap10 => SLT1_P1_050_DO06.digitalOutput_12,
    paperDirectionFlap11 => SLT1_P1_050_DO03.digitalOutput_02,
    paperDirectionFlap12 => SLT1_P1_050_DO03.digitalOutput_03,
    moveSlitterOperatorSide => SLT1_P1_050_DO04.digitalOutput_03,
    moveSlitterMotorSide => SLT1_P1_050_DO04.digitalOutput_02,
    moveSlitterOperatorSideLamp => SLT1_P1_050_DO05.digitalOutput_10,
    moveSlitterMotorSideLamp => SLT1_P1_050_DO05.digitalOutput_09,
    paperTrimOperatorSideOpen => SLT1_P1_050_DO03.digitalOutput_14,
    paperTrimOperatorSideClose => SLT1_P1_050_DO03.digitalOutput_15,
    paperTrimMotorSideOpen => SLT1_P1_050_DO03.digitalOutput_16,
    paperTrimMotorSideClose => SLT1_P1_050_DO04.digitalOutput_01,
    scorerHeightInc => SLT1_P1_050_DO03.digitalOutput_06,
    scorerHeightDec => SLT1_P1_050_DO03.digitalOutput_07,
    scorerHeightMotorStart => SLT1_P1_050_DO04.digitalOutput_04,
    scorerHeightMotorSlow => SLT1_P1_050_DO04.digitalOutput_06,
    scorerHeightMotorFast => SLT1_P1_050_DO04.digitalOutput_05,
    scorerTypeWLamp => SLT1_P1_050_DO03.digitalOutput_10,
    scorerTypeNLamp => SLT1_P1_050_DO03.digitalOutput_11,
    scorerTypeDLamp => SLT1_P1_050_DO03.digitalOutput_12,
    tractionEnabledLamp => SLT1_P1_050_DO05.digitalOutput_11,
    knifeMotorStart => SLT1_P1_050_DO02.digitalOutput_05,
    scorerMotorStart => SLT1_P1_050_DO02.digitalOutput_06,
    startExhaustMotor => SLT1_P1_050_DO05.digitalOutput_15,
    startExhaustMotorLamp => SLT1_P1_050_DO05.digitalOutput_13,
    arrKnifeRunningMetersForSharpening => hmiStatus.arrKnifeRunningMetersForSharpening,
    arrKnifeRunningMetersForLubfrication => hmiStatus.arrKnifeRunningMetersForLubfrication); // FB_SlitterControl
END_ACTION

END_PROGRAM

(* stored: Version 1.1.0.1
   POU MAIN: Id {bcc5f24d-e98e-4f1e-8506-ae85e970a150}, SpecialFunc None
   Method _00_UpdateHardware: Id {e4c53ce6-fd8e-4127-bdb2-fce90e3642e3}
   Method _01_SlitterControl: Id {b9d39506-60b6-4458-8ed3-4ff76d217975}
   Method _02_RotaryKnifeControl: Id {68d85360-836d-49fd-ad57-f50f3078e507}
   Method _04_AutomaticOrderChange: Id {bca4df97-1f1d-484b-a5f0-6669fe760ff1}
   Method _05_LineControl: Id {0e991049-e3a2-4c9d-9da8-1552c23bfe9e}
   Method _06_AlarmsControl: Id {93e274c0-7e24-4e00-974b-fae5b4347337}
   Method _07_LowerStackerControl: Id {ded993a9-e0d2-4970-9ac4-c5614fa7a4bb}
   Method _08_UpperStackerControl: Id {e9fa4f32-63bc-4e51-9bb1-e5b3ee6fc3c7}
   Action ACT_Slitter1Control: Id {1ddfe74d-250b-4331-a60d-eebef432c707} *)
